KUKA KRL program: MyProgram_233().src

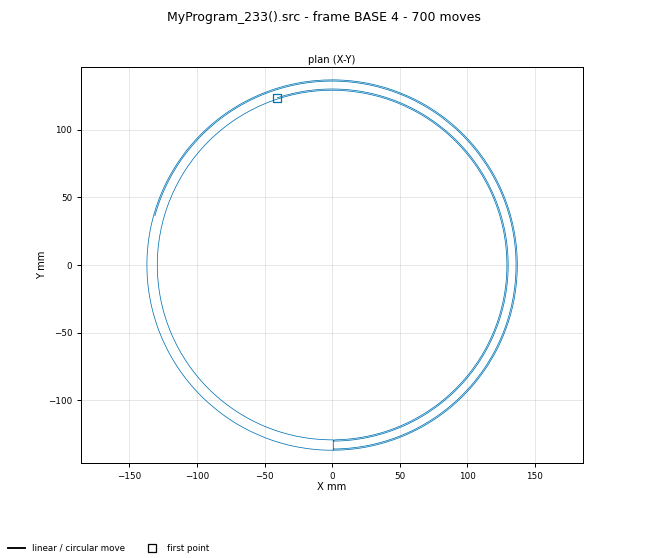
[picture p0: tool path of MyProgram_233().src in frame BASE 4, 700 of 700 moves have a stored position in this frame; points joined in program order, loops and branches not executed]
&ACCESS RVP
&REL 1
&PARAM TEMPLATE = C:\KRC\Roboter\Template\vorgabe
&PARAM EDITMASK = *
DEF MyProgram_233()
; ---- Setting reference (Base) ----
$BASE = BASE_DATA[4]

; --------------------------
; ---- Setting tool (TCP) ----
$TOOL = TOOL_DATA[3]
; --------------------------

$VEL.CP = VEL_APROX_PRINT
Startdeposition()
$VEL.CP = VEL_PRINT
LIN {X -40.5108,Y 123.8433,Z 158,A 106.7775,B 14.7751,C -0.259,E1 14.7289,E2 342.7672} C_DIS
LIN {X -37.5996,Y 124.7574,Z 158,A 105.4506,B 14.7751,C -0.2607,E1 14.7325,E2 344.0912} C_DIS
LIN {X -34.4379,Y 125.6675,Z 158,A 103.7953,B 14.7751,C -0.2561,E1 14.737,E2 345.7693} C_DIS
LIN {X -29.1894,Y 126.9876,Z 158,A 101.8109,B 14.7749,C -0.2693,E1 14.7422,E2 347.7066} C_DIS
LIN {X -26.9953,Y 127.473,Z 158,A 99.6139,B 14.7755,C -0.2357,E1 14.7486,E2 350.0402} C_DIS
LIN {X -20.6157,Y 128.6597,Z 158,A 97.7593,B 14.775,C -0.2658,E1 14.7534,E2 351.7799} C_DIS
LIN {X -13.8729,Y 129.5586,Z 158,A 94.7545,B 14.775,C -0.2668,E1 14.7617,E2 354.7844} C_DIS
LIN {X -10.0346,Y 129.9135,Z 158,A 93.1039,B 14.775,C -0.2686,E1 14.7663,E2 356.429} C_DIS
LIN {X -7.5089,Y 130.0837,Z 158,A 91.77,B 14.775,C -0.2625,E1 14.7701,E2 357.7876} C_DIS
LIN {X -2.8494,Y 130.27,Z 158,A 89.7989,B 14.775,C -0.2652,E1 14.7755,E2 359.7485} C_DIS
LIN {X 0.2302,Y 130.3001,Z 158,A 88.4188,B 14.775,C -0.2646,E1 14.7794,E2 361.131} C_DIS
LIN {X 4.1339,Y 130.2348,Z 158,A 86.7754,B 14.775,C -0.2668,E1 14.784,E2 362.7652} C_DIS
LIN {X 7.9856,Y 130.0543,Z 158,A 85.0604,B 14.775,C -0.2661,E1 14.7888,E2 364.4816} C_DIS
LIN {X 11.5872,Y 129.7845,Z 158,A 83.5435,B 14.775,C -0.268,E1 14.793,E2 365.9898} C_DIS
LIN {X 14.7399,Y 129.4647,Z 158,A 81.5298,B 14.7752,C -0.2493,E1 14.7987,E2 368.0739} C_DIS
LIN {X 19.1993,Y 128.8782,Z 158,A 80.1893,B 14.7749,C -0.2675,E1 14.8023,E2 369.341} C_DIS
LIN {X 22.8847,Y 128.2737,Z 158,A 78.3564,B 14.775,C -0.2612,E1 14.8073,E2 371.1953} C_DIS
LIN {X 27.0473,Y 127.4618,Z 158,A 76.5376,B 14.775,C -0.2616,E1 14.8123,E2 373.0085} C_DIS
LIN {X 30.989,Y 126.5612,Z 158,A 74.8488,B 14.775,C -0.2632,E1 14.8169,E2 374.6867} C_DIS
LIN {X 34.4256,Y 125.6709,Z 158,A 73.0922,B 14.7751,C -0.2562,E1 14.8217,E2 376.4656} C_DIS
LIN {X 37.7415,Y 124.7139,Z 158,A 71.8178,B 14.7751,C -0.2624,E1 14.825,E2 377.7118} C_DIS
LIN {X 41.1053,Y 123.6453,Z 158,A 70.2161,B 14.7751,C -0.2596,E1 14.8293,E2 379.3191} C_DIS
LIN {X 45.0082,Y 122.2809,Z 158,A 68.4489,B 14.7751,C -0.2595,E1 14.8339,E2 381.0806} C_DIS
LIN {X 47.9326,Y 121.1646,Z 158,A 67.0589,B 14.7751,C -0.2577,E1 14.8375,E2 382.4721} C_DIS
LIN {X 51.5684,Y 119.6599,Z 158,A 65.3226,B 14.7751,C -0.2556,E1 14.842,E2 384.2091} C_DIS
LIN {X 54.5031,Y 118.3521,Z 158,A 63.7925,B 14.7752,C -0.2504,E1 14.8459,E2 385.7528} C_DIS
LIN {X 58.0846,Y 116.637,Z 158,A 62.2133,B 14.7752,C -0.2534,E1 14.8498,E2 387.3129} C_DIS
LIN {X 60.819,Y 115.2341,Z 158,A 60.796,B 14.7752,C -0.2496,E1 14.8534,E2 388.738} C_DIS
LIN {X 63.7715,Y 113.6287,Z 158,A 59.2585,B 14.7753,C -0.2457,E1 14.8571,E2 390.2827} C_DIS
LIN {X 67.0742,Y 111.7117,Z 158,A 57.6957,B 14.7753,C -0.2469,E1 14.8609,E2 391.8325} C_DIS
LIN {X 70.2806,Y 109.722,Z 158,A 55.9342,B 14.7753,C -0.2412,E1 14.8651,E2 393.6062} C_DIS
LIN {X 74.0762,Y 107.1968,Z 158,A 54.0892,B 14.7753,C -0.2429,E1 14.8693,E2 395.4333} C_DIS
LIN {X 76.3123,Y 105.6161,Z 158,A 52.7396,B 14.7755,C -0.2364,E1 14.8724,E2 396.8001} C_DIS
LIN {X 83.8311,Y 99.7529,Z 158,A 48.7733,B 14.7755,C -0.2359,E1 14.8811,E2 400.7419} C_DIS
LIN {X 87.1361,Y 96.8796,Z 158,A 46.7285,B 14.7755,C -0.2285,E1 14.8854,E2 402.8014} C_DIS
LIN {X 90.1084,Y 94.121,Z 158,A 44.9408,B 14.7756,C -0.2248,E1 14.889,E2 404.5904} C_DIS
LIN {X 93.1997,Y 91.0613,Z 158,A 42.1103,B 14.7761,C -0.1919,E1 14.8947,E2 407.5274} C_DIS
LIN {X 97.7522,Y 86.1558,Z 158,A 40.368,B 14.7756,C -0.2235,E1 14.8977,E2 409.1333} C_DIS
LIN {X 99.829,Y 83.7404,Z 158,A 38.7374,B 14.7758,C -0.213,E1 14.9007,E2 410.7915} C_DIS
LIN {X 102.3423,Y 80.6497,Z 158,A 36.9316,B 14.7758,C -0.2073,E1 14.9039,E2 412.6046} C_DIS
LIN {X 105.1336,Y 76.9756,Z 158,A 35.0273,B 14.7758,C -0.2065,E1 14.9071,E2 414.4959} C_DIS
LIN {X 107.1572,Y 74.1333,Z 158,A 33.457,B 14.776,C -0.2017,E1 14.9096,E2 416.0716} C_DIS
LIN {X 109.47,Y 70.6733,Z 158,A 31.6182,B 14.776,C -0.1969,E1 14.9124,E2 417.9127} C_DIS
LIN {X 111.7477,Y 67.0138,Z 158,A 29.7051,B 14.776,C -0.1916,E1 14.9152,E2 419.8294} C_DIS
LIN {X 113.64,Y 63.7515,Z 158,A 28.0795,B 14.7761,C -0.1884,E1 14.9174,E2 421.4526} C_DIS
LIN {X 115.5412,Y 60.2341,Z 158,A 26.3549,B 14.7761,C -0.1849,E1 14.9197,E2 423.1746} C_DIS
LIN {X 117.1122,Y 57.1213,Z 158,A 24.9494,B 14.7761,C -0.1849,E1 14.9214,E2 424.5666} C_DIS
LIN {X 118.4334,Y 54.3273,Z 158,A 23.5787,B 14.7762,C -0.1809,E1 14.9231,E2 425.9399} C_DIS
LIN {X 119.9368,Y 50.927,Z 158,A 21.9716,B 14.7762,C -0.1774,E1 14.9248,E2 427.5454} C_DIS
LIN {X 121.0941,Y 48.1087,Z 158,A 20.662,B 14.7762,C -0.1747,E1 14.9262,E2 428.8527} C_DIS
LIN {X 122.0988,Y 45.4943,Z 158,A 19.4496,B 14.7763,C -0.1719,E1 14.9274,E2 430.0639} C_DIS
LIN {X 123.1367,Y 42.6048,Z 158,A 18.0772,B 14.7763,C -0.1674,E1 14.9287,E2 431.4403} C_DIS
LIN {X 124.1541,Y 39.5421,Z 158,A 16.6266,B 14.7764,C -0.1623,E1 14.9299,E2 432.896} C_DIS
LIN {X 125.2221,Y 36.0224,Z 158,A 15.079,B 14.7764,C -0.16,E1 14.9312,E2 434.4372} C_DIS
LIN {X 126.1859,Y 32.4831,Z 158,A 13.215,B 14.7766,C -0.1471,E1 14.9325,E2 436.3323} C_DIS
LIN {X 127.3684,Y 27.4799,Z 158,A 10.9043,B 14.7766,C -0.1389,E1 14.9339,E2 438.6511} C_DIS
LIN {X 128.028,Y 24.2226,Z 158,A 9.7326,B 14.7766,C -0.1441,E1 14.9345,E2 439.7907} C_DIS
LIN {X 128.6085,Y 20.928,Z 158,A 7.975,B 14.7767,C -0.1304,E1 14.9354,E2 441.5834} C_DIS
LIN {X 129.1193,Y 17.5046,Z 158,A 6.6957,B 14.7767,C -0.1338,E1 14.9358,E2 442.8361} C_DIS
LIN {X 129.5993,Y 13.4944,Z 158,A 5.074,B 14.7767,C -0.1336,E1 14.9363,E2 444.4418} C_DIS
LIN {X 129.9364,Y 9.7203,Z 158,A 3.3807,B 14.7767,C -0.1277,E1 14.9367,E2 446.1402} C_DIS
LIN {X 130.1635,Y 5.9747,Z 158,A 1.6403,B 14.7768,C -0.1198,E1 14.937,E2 447.8932} C_DIS
LIN {X 130.2801,Y 2.244,Z 158,A 0.1423,B 14.7768,C -0.1196,E1 14.937,E2 449.3764} C_DIS
LIN {X 130.2859,Y -1.8955,Z 158,A -1.6435,B 14.7768,C -0.1152,E1 14.937,E2 451.1603} C_DIS
LIN {X 130.19,Y -5.3434,Z 158,A -3.2527,B 14.7769,C -0.1076,E1 14.937,E2 452.7822} C_DIS
LIN {X 129.9186,Y -9.9649,Z 158,A -5.9348,B 14.7771,C -0.0802,E1 14.9364,E2 455.5425} C_DIS
LIN {X 129.3731,Y -15.5074,Z 158,A -7.5578,B 14.777,C -0.1,E1 14.9359,E2 457.0719} C_DIS
LIN {X 129.005,Y -18.3195,Z 158,A -9.5341,B 14.7771,C -0.0723,E1 14.9351,E2 459.1353} C_DIS
LIN {X 128.1366,Y -23.6512,Z 158,A -11.1383,B 14.7771,C -0.0905,E1 14.9343,E2 460.6523} C_DIS
LIN {X 127.2398,Y -28.0756,Z 158,A -13.1387,B 14.7771,C -0.0841,E1 14.9332,E2 462.6571} C_DIS
LIN {X 126.2536,Y -32.2163,Z 158,A -15.0385,B 14.7771,C -0.0776,E1 14.9319,E2 464.5625} C_DIS
LIN {X 124.8734,Y -37.2135,Z 158,A -17.2259,B 14.7771,C -0.0739,E1 14.9302,E2 466.7422} C_DIS
LIN {X 123.7298,Y -40.8516,Z 158,A -18.9168,B 14.7771,C -0.0686,E1 14.9288,E2 468.4368} C_DIS
LIN {X 122.6296,Y -44.0434,Z 158,A -21.7356,B 14.7773,C -0.0208,E1 14.926,E2 471.4133} C_DIS
LIN {X 119.44,Y -52.0772,Z 158,A -24.233,B 14.7773,C -0.0524,E1 14.9234,E2 473.7638} C_DIS
LIN {X 116.7284,Y -57.8993,Z 158,A -27.0512,B 14.7773,C -0.0448,E1 14.92,E2 476.585} C_DIS
LIN {X 114.986,Y -61.2914,Z 158,A -28.6247,B 14.7773,C -0.0436,E1 14.918,E2 478.1486} C_DIS
LIN {X 112.9775,Y -64.9195,Z 158,A -30.4029,B 14.7773,C -0.0402,E1 14.9156,E2 479.9238} C_DIS
LIN {X 110.9729,Y -68.2886,Z 158,A -32.0131,B 14.7773,C -0.0393,E1 14.9133,E2 481.5227} C_DIS
LIN {X 109.6462,Y -70.3989,Z 158,A -33.112,B 14.7773,C -0.0363,E1 14.9116,E2 482.6234} C_DIS
LIN {X 108.2654,Y -72.5046,Z 158,A -34.3195,B 14.7773,C -0.0302,E1 14.9097,E2 483.8442} C_DIS
LIN {X 105.9657,Y -75.8258,Z 158,A -36.2678,B 14.7773,C -0.0201,E1 14.9066,E2 485.8151} C_DIS
LIN {X 103.7855,Y -78.7844,Z 158,A -37.7168,B 14.7773,C -0.0215,E1 14.9042,E2 487.2465} C_DIS
LIN {X 101.3531,Y -81.8892,Z 158,A -39.4296,B 14.7773,C -0.0179,E1 14.9012,E2 488.9589} C_DIS
LIN {X 98.3316,Y -85.494,Z 158,A -41.7666,B 14.7773,C -0.0043,E1 14.8969,E2 491.3301} C_DIS
LIN {X 96.0761,Y -88.0211,Z 158,A -42.911,B 14.7773,C -0.012,E1 14.8948,E2 492.4356} C_DIS
LIN {X 93.3589,Y -90.8985,Z 158,A -44.7247,B 14.7773,C -0.0056,E1 14.8913,E2 494.2602} C_DIS
LIN {X 89.4912,Y -94.7081,Z 158,A -47.1654,B 14.7773,C 0.0013,E1 14.8864,E2 496.71} C_DIS
LIN {X 86.752,Y -97.2236,Z 158,A -48.7508,B 14.7773,C 0.0032,E1 14.8831,E2 498.2915} C_DIS
LIN {X 83.627,Y -99.9241,Z 158,A -50.4995,B 14.7773,C 0.0048,E1 14.8794,E2 500.0343} C_DIS
LIN {X 80.0007,Y -102.8504,Z 158,A -52.3931,B 14.7773,C 0.0039,E1 14.8753,E2 501.9119} C_DIS
LIN {X 78.0349,Y -104.3499,Z 158,A -53.5757,B 14.7773,C 0.0091,E1 14.8726,E2 503.107} C_DIS
LIN {X 75.6115,Y -106.119,Z 158,A -54.8753,B 14.7773,C 0.0109,E1 14.8697,E2 504.4058} C_DIS
LIN {X 72.5816,Y -108.214,Z 158,A -56.3904,B 14.7773,C 0.0105,E1 14.8662,E2 505.9102} C_DIS
LIN {X 70.5262,Y -109.5648,Z 158,A -57.4656,B 14.7773,C 0.0122,E1 14.8637,E2 506.9858} C_DIS
LIN {X 67.235,Y -111.6145,Z 158,A -59.2828,B 14.7773,C 0.0187,E1 14.8593,E2 508.8182} C_DIS
LIN {X 63.65,Y -113.697,Z 158,A -61.5059,B 14.7773,C 0.0343,E1 14.8538,E2 511.0903} C_DIS
LIN {X 60.2129,Y -115.5523,Z 158,A -63.3497,B 14.7773,C 0.0409,E1 14.8492,E2 512.9505} C_DIS
LIN {X 56.033,Y -117.6355,Z 158,A -64.8162,B 14.7773,C 0.0254,E1 14.8457,E2 514.3499} C_DIS
LIN {X 52.9667,Y -119.0478,Z 158,A -66.328,B 14.7773,C 0.0283,E1 14.8418,E2 515.8664} C_DIS
LIN {X 49.793,Y -120.4103,Z 158,A -67.7428,B 14.7773,C 0.027,E1 14.8382,E2 517.2703} C_DIS
LIN {X 46.482,Y -121.7285,Z 158,A -69.3474,B 14.7773,C 0.0302,E1 14.834,E2 518.8807} C_DIS
LIN {X 43.6924,Y -122.7561,Z 158,A -70.6467,B 14.7773,C 0.0314,E1 14.8306,E2 520.1802} C_DIS
LIN {X 37.793,Y -124.6982,Z 158,A -73.2996,B 14.7773,C 0.0319,E1 14.8236,E2 522.8262} C_DIS
LIN {X 34.1254,Y -125.7522,Z 158,A -74.9414,B 14.7773,C 0.0324,E1 14.8192,E2 524.465} C_DIS
LIN {X 31.4215,Y -126.4553,Z 158,A -76.5158,B 14.7773,C 0.0442,E1 14.8148,E2 526.0813} C_DIS
LIN {X 24.1591,Y -128.0402,Z 158,A -79.544,B 14.7773,C 0.0393,E1 14.8066,E2 529.0834} C_DIS
LIN {X 21.0197,Y -128.5932,Z 158,A -80.9175,B 14.7773,C 0.0393,E1 14.8028,E2 530.4546} C_DIS
LIN {X 17.736,Y -129.0883,Z 158,A -82.5197,B 14.7773,C 0.0446,E1 14.7983,E2 532.0746} C_DIS
LIN {X 13.8148,Y -129.5649,Z 158,A -84.1828,B 14.7773,C 0.0432,E1 14.7937,E2 533.73} C_DIS
LIN {X 9.1695,Y -129.9766,Z 158,A -86.2845,B 14.7773,C 0.0455,E1 14.7879,E2 535.8389} C_DIS
LIN {X 5.0148,Y -130.2028,Z 158,A -88.0308,B 14.7773,C 0.0436,E1 14.783,E2 537.5764} C_DIS
LIN {X 0.9154,Y -130.2963,Z 158,A -89.8605,B 14.7773,C 0.0447,E1 14.7779,E2 539.4102} C_DIS
Enddeposition()
LIN {X 0.9154,Y -130.2963,Z 158,A -89.8605,B 14.7773,C 0.0447,E1 14.7779,E2 539.4102} C_DIS
Startdeposition()
$VEL.CP = VEL_PRINT
LIN {X 1.8704,Y -129.3568,Z 158,A -88.8345,B 14.7779,C 0.0171,E1 14.7817,E2 538.2762} C_DIS
LIN {X 5.0391,Y -129.2718,Z 158,A -87.4155,B 14.7779,C 0.0163,E1 14.7857,E2 536.8546} C_DIS
LIN {X 7.9326,Y -129.1265,Z 158,A -86.0775,B 14.7779,C 0.0142,E1 14.7894,E2 535.5095} C_DIS
LIN {X 11.1084,Y -128.8923,Z 158,A -84.6755,B 14.7779,C 0.0139,E1 14.7933,E2 534.1076} C_DIS
LIN {X 14.2559,Y -128.5827,Z 158,A -83.1246,B 14.7779,C 0.0087,E1 14.7977,E2 532.538} C_DIS
LIN {X 17.4162,Y -128.1936,Z 158,A -81.876,B 14.7779,C 0.0129,E1 14.8011,E2 531.3078} C_DIS
LIN {X 20.566,Y -127.7268,Z 158,A -80.3675,B 14.7779,C 0.009,E1 14.8053,E2 529.7867} C_DIS
LIN {X 24.2361,Y -127.0793,Z 158,A -78.992,B 14.7779,C 0.0163,E1 14.809,E2 528.4426} C_DIS
LIN {X 26.7211,Y -126.5815,Z 158,A -77.7134,B 14.7779,C 0.0107,E1 14.8125,E2 527.1448} C_DIS
LIN {X 29.9082,Y -125.8658,Z 158,A -76.181,B 14.7779,C 0.0068,E1 14.8167,E2 525.601} C_DIS
LIN {X 33.2672,Y -125.0192,Z 158,A -74.8008,B 14.7779,C 0.0102,E1 14.8204,E2 524.2379} C_DIS
LIN {X 36.0209,Y -124.2542,Z 158,A -73.4572,B 14.7779,C 0.0065,E1 14.824,E2 522.884} C_DIS
LIN {X 39.0482,Y -123.3363,Z 158,A -72.0632,B 14.7779,C 0.0053,E1 14.8278,E2 521.4897} C_DIS
LIN {X 42.4611,Y -122.2029,Z 158,A -70.5633,B 14.7779,C 0.0064,E1 14.8317,E2 519.9994} C_DIS
LIN {X 45.0721,Y -121.2646,Z 158,A -69.2472,B 14.7779,C 0.0023,E1 14.8352,E2 518.672} C_DIS
LIN {X 48.0423,Y -120.1189,Z 158,A -67.8483,B 14.7779,C 0.0008,E1 14.8388,E2 517.273} C_DIS
LIN {X 50.972,Y -118.9054,Z 158,A -66.4449,B 14.7779,C -0.001,E1 14.8424,E2 515.8685} C_DIS
LIN {X 53.8674,Y -117.6222,Z 158,A -65.063,B 14.7779,C -0.0022,E1 14.8459,E2 514.4877} C_DIS
LIN {X 56.6975,Y -116.285,Z 158,A -63.6928,B 14.7779,C -0.0037,E1 14.8494,E2 513.1181} C_DIS
LIN {X 59.4453,Y -114.9057,Z 158,A -62.3199,B 14.7779,C -0.0061,E1 14.8528,E2 511.7426} C_DIS
LIN {X 62.4679,Y -113.2907,Z 158,A -60.7953,B 14.7779,C -0.0087,E1 14.8566,E2 510.2156} C_DIS
LIN {X 65.1434,Y -111.7741,Z 158,A -59.4503,B 14.7779,C -0.0104,E1 14.8598,E2 508.8712} C_DIS
LIN {X 68.4953,Y -109.7515,Z 158,A -57.8772,B 14.7779,C -0.0082,E1 14.8635,E2 507.3155} C_DIS
LIN {X 70.5632,Y -108.4335,Z 158,A -56.6501,B 14.7779,C -0.0146,E1 14.8664,E2 506.0704} C_DIS
LIN {X 73.1984,Y -106.6722,Z 158,A -55.2581,B 14.7779,C -0.0168,E1 14.8697,E2 504.6782} C_DIS
LIN {X 75.7896,Y -104.8472,Z 158,A -53.8699,B 14.7779,C -0.0189,E1 14.8728,E2 503.2903} C_DIS
LIN {X 78.9589,Y -102.4822,Z 158,A -51.9922,B 14.7779,C -0.0264,E1 14.877,E2 501.3956} C_DIS
LIN {X 82.0782,Y -100.001,Z 158,A -50.2104,B 14.7779,C -0.0305,E1 14.8809,E2 499.6098} C_DIS
LIN {X 85.6925,Y -96.9214,Z 158,A -48.1287,B 14.7779,C -0.0342,E1 14.8853,E2 497.5282} C_DIS
LIN {X 89.1886,Y -93.7146,Z 158,A -46.1035,B 14.7779,C -0.0363,E1 14.8894,E2 495.5096} C_DIS
LIN {X 92.0419,Y -90.9142,Z 158,A -44.279,B 14.7779,C -0.042,E1 14.893,E2 493.6765} C_DIS
LIN {X 95.313,Y -87.478,Z 158,A -42.2006,B 14.7779,C -0.0461,E1 14.897,E2 491.5983} C_DIS
LIN {X 98.4499,Y -83.9322,Z 158,A -40.2684,B 14.7779,C -0.0457,E1 14.9005,E2 489.6831} C_DIS
LIN {X 101.0061,Y -80.8384,Z 158,A -38.36,B 14.7779,C -0.0543,E1 14.9039,E2 487.7568} C_DIS
LIN {X 103.901,Y -77.0817,Z 158,A -36.4277,B 14.7779,C -0.054,E1 14.9071,E2 485.8419} C_DIS
LIN {X 105.7745,Y -74.4898,Z 158,A -35.026,B 14.7779,C -0.0571,E1 14.9094,E2 484.4401} C_DIS
LIN {X 107.5679,Y -71.8758,Z 158,A -33.6347,B 14.7778,C -0.0603,E1 14.9116,E2 483.0485} C_DIS
LIN {X 109.2967,Y -69.2188,Z 158,A -32.2315,B 14.7778,C -0.0639,E1 14.9137,E2 481.6435} C_DIS
LIN {X 110.9657,Y -66.5108,Z 158,A -30.8514,B 14.7778,C -0.0667,E1 14.9157,E2 480.265} C_DIS
LIN {X 112.5675,Y -63.7628,Z 158,A -29.4479,B 14.7778,C -0.0703,E1 14.9176,E2 478.8604} C_DIS
LIN {X 114.1018,Y -60.974,Z 158,A -28.0337,B 14.7778,C -0.0743,E1 14.9195,E2 477.4438} C_DIS
LIN {X 115.5605,Y -58.1599,Z 158,A -26.5379,B 14.7778,C -0.0812,E1 14.9214,E2 475.9351} C_DIS
LIN {X 116.9596,Y -55.2918,Z 158,A -25.208,B 14.7777,C -0.0824,E1 14.923,E2 474.6133} C_DIS
LIN {X 118.2696,Y -52.4305,Z 158,A -23.8839,B 14.7777,C -0.084,E1 14.9245,E2 473.2957} C_DIS
LIN {X 119.5144,Y -49.5268,Z 158,A -22.4999,B 14.7777,C -0.0874,E1 14.926,E2 471.9116} C_DIS
LIN {X 120.6905,Y -46.5873,Z 158,A -21.1146,B 14.7777,C -0.0909,E1 14.9275,E2 470.5265} C_DIS
LIN {X 121.8119,Y -43.5713,Z 158,A -19.7027,B 14.7777,C -0.0946,E1 14.9288,E2 469.1143} C_DIS
LIN {X 122.8405,Y -40.5809,Z 158,A -18.3158,B 14.7777,C -0.0982,E1 14.93,E2 467.7271} C_DIS
LIN {X 123.798,Y -37.5587,Z 158,A -16.9229,B 14.7776,C -0.1019,E1 14.9312,E2 466.3337} C_DIS
LIN {X 124.6862,Y -34.4963,Z 158,A -15.4594,B 14.7776,C -0.1077,E1 14.9323,E2 464.8624} C_DIS
LIN {X 125.6787,Y -30.6845,Z 158,A -13.9628,B 14.7776,C -0.1047,E1 14.9333,E2 463.3928} C_DIS
LIN {X 126.2253,Y -28.3536,Z 158,A -12.7571,B 14.7775,C -0.1126,E1 14.9341,E2 462.1686} C_DIS
LIN {X 126.9119,Y -25.1076,Z 158,A -11.3092,B 14.7775,C -0.1163,E1 14.9349,E2 460.7213} C_DIS
LIN {X 127.464,Y -22.1343,Z 158,A -9.9823,B 14.7775,C -0.1199,E1 14.9355,E2 459.3942} C_DIS
LIN {X 127.9772,Y -18.9423,Z 158,A -8.5548,B 14.7775,C -0.124,E1 14.9362,E2 457.9653} C_DIS
LIN {X 128.394,Y -15.8699,Z 158,A -7.2017,B 14.7774,C -0.1275,E1 14.9366,E2 456.6129} C_DIS
LIN {X 128.732,Y -12.8404,Z 158,A -5.8713,B 14.7774,C -0.1309,E1 14.937,E2 455.283} C_DIS
LIN {X 129.0205,Y -9.5023,Z 158,A -4.391,B 14.7774,C -0.1353,E1 14.9374,E2 453.8013} C_DIS
LIN {X 129.2548,Y -5.4753,Z 158,A -2.5487,B 14.7772,C -0.1425,E1 14.9376,E2 451.9502} C_DIS
LIN {X 129.3623,Y -1.5416,Z 158,A -0.9468,B 14.7772,C -0.1431,E1 14.9377,E2 450.3629} C_DIS
LIN {X 129.3615,Y 1.5923,Z 158,A 0.493,B 14.7772,C -0.149,E1 14.9377,E2 448.9152} C_DIS
LIN {X 129.2822,Y 4.773,Z 158,A 2.0333,B 14.7771,C -0.1576,E1 14.9375,E2 447.3576} C_DIS
LIN {X 129.0371,Y 9.2755,Z 158,A 3.8932,B 14.7771,C -0.159,E1 14.9372,E2 445.5116} C_DIS
LIN {X 128.7458,Y 12.6969,Z 158,A 5.4984,B 14.7771,C -0.1664,E1 14.9368,E2 443.8947} C_DIS
LIN {X 128.3979,Y 15.837,Z 158,A 6.7268,B 14.7771,C -0.1649,E1 14.9364,E2 442.6848} C_DIS
LIN {X 127.9661,Y 19.02,Z 158,A 8.1441,B 14.777,C -0.1689,E1 14.9358,E2 441.2666} C_DIS
LIN {X 127.4679,Y 22.1126,Z 158,A 9.5203,B 14.777,C -0.1726,E1 14.9352,E2 439.8902} C_DIS
LIN {X 126.8921,Y 25.2051,Z 158,A 10.8943,B 14.7769,C -0.1761,E1 14.9345,E2 438.5168} C_DIS
LIN {X 126.2078,Y 28.4299,Z 158,A 12.272,B 14.7769,C -0.1777,E1 14.9337,E2 437.1471} C_DIS
LIN {X 125.489,Y 31.451,Z 158,A 13.7046,B 14.7769,C -0.1835,E1 14.9327,E2 435.7064} C_DIS
LIN {X 124.6841,Y 34.5036,Z 158,A 15.2093,B 14.7767,C -0.1911,E1 14.9316,E2 434.1876} C_DIS
LIN {X 123.7981,Y 37.5584,Z 158,A 16.4848,B 14.7767,C -0.1907,E1 14.9306,E2 432.9264} C_DIS
LIN {X 122.8363,Y 40.5934,Z 158,A 17.9865,B 14.7767,C -0.1977,E1 14.9293,E2 431.4124} C_DIS
LIN {X 121.8029,Y 43.5963,Z 158,A 19.2664,B 14.7767,C -0.1975,E1 14.9281,E2 430.1461} C_DIS
LIN {X 120.6965,Y 46.5719,Z 158,A 20.6608,B 14.7766,C -0.201,E1 14.9267,E2 428.7516} C_DIS
LIN {X 119.518,Y 49.5181,Z 158,A 22.052,B 14.7766,C -0.2044,E1 14.9253,E2 427.3608} C_DIS
LIN {X 118.2648,Y 52.4412,Z 158,A 23.4461,B 14.7765,C -0.2078,E1 14.9237,E2 425.9671} C_DIS
LIN {X 116.9451,Y 55.3221,Z 158,A 24.8349,B 14.7765,C -0.2111,E1 14.9221,E2 424.5787} C_DIS
LIN {X 115.5543,Y 58.1721,Z 158,A 26.2245,B 14.7765,C -0.2143,E1 14.9203,E2 423.1897} C_DIS
LIN {X 113.9971,Y 61.1689,Z 158,A 27.6625,B 14.7764,C -0.2163,E1 14.9185,E2 421.7571} C_DIS
LIN {X 112.5602,Y 63.7755,Z 158,A 29.0181,B 14.7764,C -0.2209,E1 14.9166,E2 420.3962} C_DIS
LIN {X 110.9695,Y 66.5044,Z 158,A 30.4133,B 14.7763,C -0.2244,E1 14.9146,E2 419.0002} C_DIS
LIN {X 108.9939,Y 69.6944,Z 158,A 31.9443,B 14.7763,C -0.2243,E1 14.9124,E2 417.4832} C_DIS
LIN {X 107.5569,Y 71.8922,Z 158,A 33.2084,B 14.7762,C -0.2304,E1 14.9104,E2 416.2064} C_DIS
LIN {X 105.7623,Y 74.507,Z 158,A 34.5986,B 14.7762,C -0.2333,E1 14.9082,E2 414.8169} C_DIS
LIN {X 103.5733,Y 77.5218,Z 158,A 36.2797,B 14.776,C -0.2382,E1 14.9054,E2 413.131} C_DIS
LIN {X 101.0079,Y 80.8362,Z 158,A 38.24,B 14.776,C -0.2458,E1 14.902,E2 411.1573} C_DIS
LIN {X 97.9574,Y 84.5063,Z 158,A 40.175,B 14.776,C -0.2448,E1 14.8985,E2 409.2418} C_DIS
LIN {X 95.8745,Y 86.8623,Z 158,A 41.7048,B 14.7758,C -0.2522,E1 14.8957,E2 407.6953} C_DIS
LIN {X 92.6666,Y 90.2775,Z 158,A 43.7557,B 14.7758,C -0.2558,E1 14.8917,E2 405.646} C_DIS
LIN {X 89.7778,Y 93.1504,Z 158,A 45.5701,B 14.7757,C -0.2598,E1 14.8881,E2 403.8295} C_DIS
LIN {X 86.2924,Y 96.3877,Z 158,A 47.6586,B 14.7757,C -0.2633,E1 14.8838,E2 401.7421} C_DIS
LIN {X 83.298,Y 98.9871,Z 158,A 49.3903,B 14.7756,C -0.2659,E1 14.8801,E2 400.0126} C_DIS
LIN {X 79.6543,Y 101.9424,Z 158,A 51.3138,B 14.7756,C -0.2647,E1 14.8759,E2 398.1063} C_DIS
LIN {X 76.5448,Y 104.297,Z 158,A 52.8952,B 14.7756,C -0.2631,E1 14.8724,E2 396.5412} C_DIS
LIN {X 74.494,Y 105.7716,Z 158,A 54.141,B 14.7756,C -0.269,E1 14.8696,E2 395.2803} C_DIS
LIN {X 71.8789,Y 107.5658,Z 158,A 55.5369,B 14.7755,C -0.271,E1 14.8663,E2 393.885} C_DIS
LIN {X 68.5385,Y 109.7246,Z 158,A 57.4465,B 14.7754,C -0.2783,E1 14.8618,E2 391.9577} C_DIS
LIN {X 65.138,Y 111.7772,Z 158,A 59.0374,B 14.7754,C -0.2756,E1 14.858,E2 390.386} C_DIS
LIN {X 62.3796,Y 113.3396,Z 158,A 60.4418,B 14.7754,C -0.2775,E1 14.8546,E2 388.9813} C_DIS
LIN {X 59.5725,Y 114.839,Z 158,A 61.8465,B 14.7754,C -0.2793,E1 14.8511,E2 387.577} C_DIS
LIN {X 56.7398,Y 116.2642,Z 158,A 63.2428,B 14.7754,C -0.2808,E1 14.8476,E2 386.1814} C_DIS
LIN {X 53.873,Y 117.6196,Z 158,A 64.6388,B 14.7753,C -0.2822,E1 14.8441,E2 384.7862} C_DIS
LIN {X 50.6665,Y 119.0375,Z 158,A 66.1801,B 14.7753,C -0.2835,E1 14.8401,E2 383.2463} C_DIS
LIN {X 48.0346,Y 120.1219,Z 158,A 67.4419,B 14.7753,C -0.2849,E1 14.8369,E2 381.9843} C_DIS
LIN {X 45.0726,Y 121.2644,Z 158,A 68.8419,B 14.7753,C -0.2861,E1 14.8332,E2 380.5849} C_DIS
LIN {X 41.276,Y 122.609,Z 158,A 70.79,B 14.7751,C -0.2927,E1 14.828,E2 378.6179} C_DIS
LIN {X 37.5536,Y 123.7995,Z 158,A 72.3454,B 14.7751,C -0.2888,E1 14.8239,E2 377.083} C_DIS
LIN {X 34.5005,Y 124.685,Z 158,A 73.824,B 14.7751,C -0.2919,E1 14.8199,E2 375.5964} C_DIS
LIN {X 30.8477,Y 125.6393,Z 158,A 75.3196,B 14.7751,C -0.2877,E1 14.816,E2 374.1214} C_DIS
LIN {X 28.3547,Y 126.225,Z 158,A 76.543,B 14.7751,C -0.291,E1 14.8126,E2 372.888} C_DIS
LIN {X 25.2462,Y 126.8837,Z 158,A 77.9451,B 14.7751,C -0.2916,E1 14.8088,E2 371.4868} C_DIS
LIN {X 22.1444,Y 127.4622,Z 158,A 79.4205,B 14.7751,C -0.2945,E1 14.8047,E2 370.0029} C_DIS
LIN {X 18.985,Y 127.9711,Z 158,A 80.8587,B 14.7751,C -0.2957,E1 14.8007,E2 368.5626} C_DIS
LIN {X 15.883,Y 128.3924,Z 158,A 82.1755,B 14.7751,C -0.294,E1 14.7971,E2 367.2542} C_DIS
LIN {X 12.6795,Y 128.7475,Z 158,A 83.5848,B 14.7751,C -0.2938,E1 14.7932,E2 365.8475} C_DIS
LIN {X 9.5064,Y 129.0202,Z 158,A 85.1433,B 14.775,C -0.2984,E1 14.7888,E2 364.2725} C_DIS
LIN {X 5.4109,Y 129.2573,Z 158,A 86.9292,B 14.775,C -0.2976,E1 14.7838,E2 362.491} C_DIS
LIN {X 1.5855,Y 129.3616,Z 158,A 88.4775,B 14.775,C -0.2932,E1 14.7795,E2 360.9603} C_DIS
LIN {X -1.5842,Y 129.3616,Z 158,A 89.9211,B 14.775,C -0.2942,E1 14.7755,E2 359.5128} C_DIS
LIN {X -4.768,Y 129.2824,Z 158,A 91.4165,B 14.775,C -0.2964,E1 14.7713,E2 358.0083} C_DIS
LIN {X -7.9373,Y 129.1262,Z 158,A 92.719,B 14.775,C -0.2931,E1 14.7677,E2 356.7183} C_DIS
LIN {X -11.1107,Y 128.8921,Z 158,A 94.1241,B 14.775,C -0.2925,E1 14.7638,E2 355.3146} C_DIS
LIN {X -15.0056,Y 128.4971,Z 158,A 95.6793,B 14.7752,C -0.2866,E1 14.7595,E2 353.7809} C_DIS
LIN {X -17.4315,Y 128.1916,Z 158,A 96.9383,B 14.7752,C -0.2911,E1 14.756,E2 352.5025} C_DIS
LIN {X -20.558,Y 127.7281,Z 158,A 98.3577,B 14.7752,C -0.2909,E1 14.7521,E2 351.0817} C_DIS
LIN {X -23.648,Y 127.1917,Z 158,A 99.7546,B 14.7752,C -0.2903,E1 14.7482,E2 349.6849} C_DIS
LIN {X -26.8057,Y 126.5632,Z 158,A 101.1804,B 14.7752,C -0.2893,E1 14.7443,E2 348.2601} C_DIS
LIN {X -29.8929,Y 125.8695,Z 158,A 102.5896,B 14.7752,C -0.2885,E1 14.7405,E2 346.8509} C_DIS
LIN {X -32.9844,Y 125.0947,Z 158,A 104.1378,B 14.7752,C -0.2912,E1 14.7363,E2 345.2881} C_DIS
LIN {X -36.0387,Y 124.249,Z 158,A 105.4058,B 14.7752,C -0.286,E1 14.7329,E2 344.0368} C_DIS
LIN {X -39.0711,Y 123.329,Z 158,A 106.8132,B 14.7752,C -0.2848,E1 14.7292,E2 342.63} C_DIS
LIN {X -42.071,Y 122.3381,Z 158,A 108.2261,B 14.7752,C -0.2837,E1 14.7254,E2 341.2168} C_DIS
LIN {X -45.0765,Y 121.2629,Z 158,A 109.6389,B 14.7752,C -0.2821,E1 14.7217,E2 339.8053} C_DIS
LIN {X -48.0477,Y 120.1167,Z 158,A 111.0564,B 14.7753,C -0.2806,E1 14.7181,E2 338.3882} C_DIS
LIN {X -50.9916,Y 118.8969,Z 158,A 112.4639,B 14.7753,C -0.2787,E1 14.7144,E2 336.9825} C_DIS
LIN {X -53.877,Y 117.6178,Z 158,A 114.001,B 14.7753,C -0.2808,E1 14.7105,E2 335.4307} C_DIS
LIN {X -56.7409,Y 116.2636,Z 158,A 115.2781,B 14.7754,C -0.2753,E1 14.7073,E2 334.1694} C_DIS
LIN {X -59.5696,Y 114.8405,Z 158,A 116.6737,B 14.7754,C -0.2731,E1 14.7038,E2 332.7759} C_DIS
LIN {X -62.9274,Y 113.0363,Z 158,A 118.2492,B 14.7756,C -0.2674,E1 14.7,E2 331.2151} C_DIS
LIN {X -65.1416,Y 111.7752,Z 158,A 119.5345,B 14.7756,C -0.2699,E1 14.6969,E2 329.913} C_DIS
LIN {X -67.8877,Y 110.1286,Z 158,A 120.9556,B 14.7756,C -0.2677,E1 14.6935,E2 328.493} C_DIS
LIN {X -70.5661,Y 108.4316,Z 158,A 122.368,B 14.7756,C -0.2655,E1 14.6902,E2 327.0811} C_DIS
LIN {X -73.2027,Y 106.6693,Z 158,A 123.778,B 14.7756,C -0.2632,E1 14.6869,E2 325.672} C_DIS
LIN {X -76.1949,Y 104.5534,Z 158,A 125.3216,B 14.7757,C -0.258,E1 14.6834,E2 324.1393} C_DIS
LIN {X -78.9664,Y 102.4763,Z 158,A 126.956,B 14.7757,C -0.2579,E1 14.6798,E2 322.4951} C_DIS
LIN {X -82.0795,Y 100,Z 158,A 128.8942,B 14.7757,C -0.2592,E1 14.6755,E2 320.5386} C_DIS
LIN {X -85.6992,Y 96.9154,Z 158,A 131.0102,B 14.7757,C -0.2552,E1 14.6711,E2 318.424} C_DIS
LIN {X -89.2031,Y 93.7008,Z 158,A 132.9715,B 14.7759,C -0.2468,E1 14.6671,E2 316.4817} C_DIS
LIN {X -91.4858,Y 91.4739,Z 158,A 134.5617,B 14.7759,C -0.2485,E1 14.6639,E2 314.8728} C_DIS
LIN {X -94.7812,Y 88.054,Z 158,A 136.6786,B 14.7759,C -0.2441,E1 14.6598,E2 312.7569} C_DIS
LIN {X -97.9529,Y 84.5116,Z 158,A 138.6439,B 14.7761,C -0.2355,E1 14.6563,E2 310.8103} C_DIS
LIN {X -100.5113,Y 81.4526,Z 158,A 140.5743,B 14.7761,C -0.2357,E1 14.6528,E2 308.8633} C_DIS
LIN {X -102.9643,Y 78.329,Z 158,A 142.2007,B 14.7762,C -0.2278,E1 14.6501,E2 307.2543} C_DIS
LIN {X -104.8445,Y 75.7932,Z 158,A 143.7391,B 14.7762,C -0.2281,E1 14.6475,E2 305.7015} C_DIS
LIN {X -106.6807,Y 73.186,Z 158,A 145.032,B 14.7762,C -0.2213,E1 14.6455,E2 304.4241} C_DIS
LIN {X -108.4481,Y 70.5408,Z 158,A 146.4491,B 14.7763,C -0.2179,E1 14.6433,E2 303.0078} C_DIS
LIN {X -110.1463,Y 67.8588,Z 158,A 147.8684,B 14.7763,C -0.2146,E1 14.6412,E2 301.5888} C_DIS
LIN {X -112.1734,Y 64.4535,Z 158,A 149.7961,B 14.7763,C -0.2146,E1 14.6384,E2 299.6436} C_DIS
LIN {X -114.2931,Y 60.612,Z 158,A 151.6317,B 14.7765,C -0.2065,E1 14.636,E2 297.8228} C_DIS
LIN {X -115.5666,Y 58.1479,Z 158,A 152.8531,B 14.7765,C -0.2029,E1 14.6345,E2 296.6038} C_DIS
LIN {X -116.9562,Y 55.299,Z 158,A 154.2861,B 14.7765,C -0.1998,E1 14.6328,E2 295.1693} C_DIS
LIN {X -118.2711,Y 52.427,Z 158,A 155.68,B 14.7767,C -0.1958,E1 14.6312,E2 293.7778} C_DIS
LIN {X -119.5204,Y 49.5126,Z 158,A 157.0972,B 14.7767,C -0.1922,E1 14.6296,E2 292.3609} C_DIS
LIN {X -120.702,Y 46.5577,Z 158,A 158.5209,B 14.7767,C -0.1886,E1 14.6282,E2 290.9374} C_DIS
LIN {X -122.0846,Y 42.8023,Z 158,A 160.473,B 14.7767,C -0.1883,E1 14.6263,E2 288.967} C_DIS
LIN {X -123.3319,Y 39.0621,Z 158,A 162.0727,B 14.7769,C -0.1793,E1 14.625,E2 287.3864} C_DIS
LIN {X -124.2558,Y 36.0157,Z 158,A 163.5086,B 14.7769,C -0.1759,E1 14.6238,E2 285.9493} C_DIS
LIN {X -125.0984,Y 32.9704,Z 158,A 164.9094,B 14.7769,C -0.1718,E1 14.6228,E2 284.5502} C_DIS
LIN {X -125.8692,Y 29.894,Z 158,A 166.3275,B 14.7769,C -0.168,E1 14.6219,E2 283.1323} C_DIS
LIN {X -126.5663,Y 26.7914,Z 158,A 167.7485,B 14.777,C -0.1642,E1 14.621,E2 281.7118} C_DIS
LIN {X -127.1901,Y 23.6568,Z 158,A 169.1743,B 14.777,C -0.1603,E1 14.6203,E2 280.2866} C_DIS
LIN {X -127.7319,Y 20.535,Z 158,A 170.6159,B 14.7771,C -0.1571,E1 14.6196,E2 278.8424} C_DIS
LIN {X -128.1956,Y 17.4011,Z 158,A 172.0329,B 14.7771,C -0.1532,E1 14.619,E2 277.4256} C_DIS
LIN {X -128.5815,Y 14.2672,Z 158,A 173.4433,B 14.7771,C -0.1494,E1 14.6186,E2 276.0154} C_DIS
LIN {X -128.8929,Y 11.1012,Z 158,A 174.8632,B 14.7772,C -0.1454,E1 14.6182,E2 274.596} C_DIS
LIN {X -129.1369,Y 7.7639,Z 158,A 176.493,B 14.7772,C -0.1449,E1 14.6179,E2 272.9511} C_DIS
LIN {X -129.3341,Y 3.0911,Z 158,A 178.4296,B 14.7773,C -0.1351,E1 14.6177,E2 271.0326} C_DIS
LIN {X -129.3725,Y -0.0564,Z 158,A 179.8987,B 14.7773,C -0.1328,E1 14.6177,E2 269.5566} C_DIS
LIN {X -129.3312,Y -3.193,Z 158,A -178.5768,B 14.7773,C -0.1323,E1 14.6178,E2 268.0181} C_DIS
LIN {X -129.1268,Y -7.9284,Z 158,A -176.6162,B 14.7774,C -0.1223,E1 14.6181,E2 266.076} C_DIS
LIN {X -128.8938,Y -11.0916,Z 158,A -175.0886,B 14.7774,C -0.1214,E1 14.6184,E2 264.5358} C_DIS
LIN {X -128.5825,Y -14.2577,Z 158,A -173.7819,B 14.7774,C -0.1145,E1 14.6188,E2 263.2426} C_DIS
LIN {X -128.1292,Y -17.8783,Z 158,A -172.2851,B 14.7775,C -0.1065,E1 14.6194,E2 261.7614} C_DIS
LIN {X -127.7273,Y -20.5628,Z 158,A -170.9163,B 14.7775,C -0.1074,E1 14.6199,E2 260.3748} C_DIS
LIN {X -127.187,Y -23.6729,Z 158,A -169.4986,B 14.7775,C -0.1038,E1 14.6206,E2 258.9563} C_DIS
LIN {X -126.5661,Y -26.7924,Z 158,A -168.0752,B 14.7775,C -0.1001,E1 14.6214,E2 257.5328} C_DIS
LIN {X -125.8662,Y -29.9063,Z 158,A -166.6558,B 14.7776,C -0.0961,E1 14.6223,E2 256.1141} C_DIS
LIN {X -125.0945,Y -32.9849,Z 158,A -165.241,B 14.7776,C -0.0923,E1 14.6233,E2 254.6998} C_DIS
LIN {X -124.2488,Y -36.0396,Z 158,A -163.8182,B 14.7776,C -0.0888,E1 14.6244,E2 253.2763} C_DIS
LIN {X -123.2542,Y -39.3054,Z 158,A -162.3519,B 14.7776,C -0.0833,E1 14.6256,E2 251.8168} C_DIS
LIN {X -122.3321,Y -42.0884,Z 158,A -160.8555,B 14.7776,C -0.085,E1 14.627,E2 250.2987} C_DIS
LIN {X -121.2585,Y -45.0884,Z 158,A -159.5558,B 14.7777,C -0.078,E1 14.6282,E2 249.0133} C_DIS
LIN {X -120.1142,Y -48.0538,Z 158,A -158.1384,B 14.7777,C -0.0744,E1 14.6297,E2 247.5962} C_DIS
LIN {X -118.902,Y -50.9797,Z 158,A -156.7272,B 14.7777,C -0.0708,E1 14.6312,E2 246.1853} C_DIS
LIN {X -117.6239,Y -53.8638,Z 158,A -155.3152,B 14.7777,C -0.0675,E1 14.6328,E2 244.7728} C_DIS
LIN {X -116.2718,Y -56.7243,Z 158,A -153.7737,B 14.7777,C -0.0675,E1 14.6347,E2 243.2163} C_DIS
LIN {X -114.8344,Y -59.5812,Z 158,A -152.4857,B 14.7777,C -0.0604,E1 14.6363,E2 241.9445} C_DIS
LIN {X -113.3326,Y -62.3923,Z 158,A -151.0403,B 14.7778,C -0.0576,E1 14.6383,E2 240.4964} C_DIS
LIN {X -111.7683,Y -65.1535,Z 158,A -149.4663,B 14.7778,C -0.0587,E1 14.6405,E2 238.9038} C_DIS
LIN {X -110.1358,Y -67.8759,Z 158,A -148.1514,B 14.7778,C -0.0527,E1 14.6424,E2 237.6007} C_DIS
LIN {X -108.4433,Y -70.5481,Z 158,A -146.7906,B 14.7778,C -0.0481,E1 14.6444,E2 236.2456} C_DIS
LIN {X -106.687,Y -73.1768,Z 158,A -145.2278,B 14.7778,C -0.0492,E1 14.6469,E2 234.6648} C_DIS
LIN {X -104.8426,Y -75.7959,Z 158,A -143.9549,B 14.7778,C -0.0419,E1 14.649,E2 233.41} C_DIS
LIN {X -102.4737,Y -78.9698,Z 158,A -142.0209,B 14.7778,C -0.0427,E1 14.6522,E2 231.4561} C_DIS
LIN {X -99.4995,Y -82.6853,Z 158,A -140.051,B 14.7778,C -0.0342,E1 14.6557,E2 229.5037} C_DIS
LIN {X -96.9203,Y -85.6938,Z 158,A -138.1309,B 14.7778,C -0.0349,E1 14.6592,E2 227.5653} C_DIS
LIN {X -94.8495,Y -87.9807,Z 158,A -136.753,B 14.7778,C -0.0324,E1 14.6619,E2 226.1869} C_DIS
LIN {X -92.037,Y -90.9192,Z 158,A -135.0927,B 14.7778,C -0.0247,E1 14.6651,E2 224.5442} C_DIS
LIN {X -89.1959,Y -93.7076,Z 158,A -133.1577,B 14.7778,C -0.026,E1 14.669,E2 222.5899} C_DIS
LIN {X -85.6956,Y -96.9187,Z 158,A -131.0483,B 14.7779,C -0.0222,E1 14.6734,E2 220.4807} C_DIS
LIN {X -82.0858,Y -99.9948,Z 158,A -128.9405,B 14.7779,C -0.0186,E1 14.6779,E2 218.373} C_DIS
LIN {X -78.3422,Y -102.9542,Z 158,A -126.9546,B 14.7779,C -0.0113,E1 14.6822,E2 216.4029} C_DIS
LIN {X -75.7895,Y -104.8472,Z 158,A -125.5429,B 14.7779,C -0.0091,E1 14.6854,E2 214.9911} C_DIS
LIN {X -73.1938,Y -106.6754,Z 158,A -124.1099,B 14.7779,C -0.0076,E1 14.6887,E2 213.5554} C_DIS
LIN {X -70.5326,Y -108.4534,Z 158,A -122.7211,B 14.7779,C -0.0046,E1 14.6919,E2 212.1703} C_DIS
LIN {X -67.9045,Y -110.1183,Z 158,A -121.3091,B 14.7779,C -0.0036,E1 14.6953,E2 210.7546} C_DIS
LIN {X -65.1423,Y -111.7748,Z 158,A -119.8889,B 14.7779,C -0.0014,E1 14.6987,E2 209.3355} C_DIS
LIN {X -62.3811,Y -113.3388,Z 158,A -118.4706,B 14.7779,C 0.0001,E1 14.7021,E2 207.9159} C_DIS
LIN {X -59.5756,Y -114.8373,Z 158,A -117.0536,B 14.7779,C 0.0017,E1 14.7057,E2 206.498} C_DIS
LIN {X -56.7426,Y -116.2628,Z 158,A -115.6452,B 14.7779,C 0.0032,E1 14.7092,E2 205.0894} C_DIS
LIN {X -53.6915,Y -117.7036,Z 158,A -114.0023,B 14.7779,C 0.0006,E1 14.7134,E2 203.429} C_DIS
LIN {X -49.504,Y -119.5239,Z 158,A -112.1186,B 14.7779,C 0.0067,E1 14.7182,E2 201.5617} C_DIS
LIN {X -46.5492,Y -120.7053,Z 158,A -110.5626,B 14.7779,C 0.0038,E1 14.7223,E2 199.9884} C_DIS
LIN {X -41.9284,Y -122.3876,Z 158,A -108.5366,B 14.7779,C 0.0102,E1 14.7276,E2 197.9803} C_DIS
LIN {X -39.0628,Y -123.3317,Z 158,A -107.1829,B 14.7779,C 0.0107,E1 14.7312,E2 196.6243} C_DIS
LIN {X -35.5069,Y -124.4036,Z 158,A -105.5484,B 14.7779,C 0.0122,E1 14.7355,E2 194.9909} C_DIS
LIN {X -32.9776,Y -125.0965,Z 158,A -104.3719,B 14.7779,C 0.0124,E1 14.7387,E2 193.8124} C_DIS
LIN {X -29.9055,Y -125.8664,Z 158,A -102.9682,B 14.7779,C 0.0132,E1 14.7425,E2 192.4083} C_DIS
LIN {X -26.8178,Y -126.5606,Z 158,A -101.5651,B 14.7779,C 0.0138,E1 14.7464,E2 191.0048} C_DIS
LIN {X -23.1237,Y -127.2869,Z 158,A -100.0696,B 14.7779,C 0.0196,E1 14.7504,E2 189.5292} C_DIS
LIN {X -20.1829,Y -127.7864,Z 158,A -98.6872,B 14.7779,C 0.0183,E1 14.7542,E2 188.1392} C_DIS
LIN {X -17.3981,Y -128.196,Z 158,A -97.3075,B 14.7779,C 0.0147,E1 14.7581,E2 186.7434} C_DIS
LIN {X -14.2599,Y -128.5823,Z 158,A -95.9094,B 14.7779,C 0.015,E1 14.762,E2 185.3451} C_DIS
LIN {X -11.0349,Y -128.8985,Z 158,A -94.4897,B 14.7779,C 0.0156,E1 14.7659,E2 183.9266} C_DIS
LIN {X -7.9166,Y -129.1275,Z 158,A -93.1023,B 14.7779,C 0.0156,E1 14.7698,E2 182.5383} C_DIS
LIN {X -4.7503,Y -129.2831,Z 158,A -91.7054,B 14.7779,C 0.0158,E1 14.7737,E2 181.1417} C_DIS
LIN {X -1.5911,Y -129.3615,Z 158,A -90.3143,B 14.7779,C 0.0159,E1 14.7776,E2 179.7509} C_DIS
LIN {X 0.9078,Y -129.3647,Z 158,A -89.4432,B 14.7779,C 0.0228,E1 14.7799,E2 178.9071} C_DIS
Enddeposition()
LIN {X 0.9597,Y -137.0527,Z 159,A -92.8598,B 24.9713,C -1.2377,E1 25.0005,E2 179.5674} C_DIS
Startdeposition()
$VEL.CP = VEL_PRINT
LIN {X -5.2813,Y -136.9557,Z 159,A -95.4325,B 24.9713,C -1.2392,E1 24.9934,E2 182.1367} C_DIS
LIN {X -8.4201,Y -136.7985,Z 159,A -96.84,B 24.9715,C -1.2341,E1 24.9894,E2 183.5568} C_DIS
LIN {X -12.4091,Y -136.4962,Z 159,A -99.1922,B 24.9731,C -1.1978,E1 24.9826,E2 185.9961} C_DIS
LIN {X -17.8456,Y -135.8905,Z 159,A -100.435,B 24.9705,C -1.2541,E1 24.9795,E2 187.1064} C_DIS
LIN {X -24.6121,Y -134.8301,Z 159,A -103.6254,B 24.9713,C -1.2373,E1 24.9706,E2 190.3395} C_DIS
LIN {X -28.0212,Y -134.164,Z 159,A -105.2172,B 24.9716,C -1.2305,E1 24.9662,E2 191.9494} C_DIS
LIN {X -31.9677,Y -133.277,Z 159,A -106.7877,B 24.9713,C -1.2378,E1 24.962,E2 193.5045} C_DIS
LIN {X -35.4042,Y -132.4055,Z 159,A -108.2494,B 24.9713,C -1.2398,E1 24.958,E2 194.9637} C_DIS
LIN {X -38.6063,Y -131.5074,Z 159,A -109.6605,B 24.9713,C -1.2396,E1 24.9542,E2 196.3774} C_DIS
LIN {X -42.0011,Y -130.4632,Z 159,A -111.1444,B 24.9712,C -1.2408,E1 24.9503,E2 197.8611} C_DIS
LIN {X -45.5688,Y -129.2618,Z 159,A -112.7992,B 24.9713,C -1.2379,E1 24.9459,E2 199.5261} C_DIS
LIN {X -50.174,Y -127.5441,Z 159,A -114.7347,B 24.9709,C -1.2462,E1 24.9409,E2 201.446} C_DIS
LIN {X -59.4901,Y -123.4736,Z 159,A -119.0248,B 24.9708,C -1.2488,E1 24.93,E2 205.7402} C_DIS
LIN {X -62.411,Y -122.0226,Z 159,A -120.435,B 24.9708,C -1.2481,E1 24.9264,E2 207.1557} C_DIS
LIN {X -65.7883,Y -120.2375,Z 159,A -122.0656,B 24.9708,C -1.2485,E1 24.9224,E2 208.79} C_DIS
LIN {X -69.2875,Y -118.2556,Z 159,A -123.7412,B 24.9707,C -1.2512,E1 24.9183,E2 210.4641} C_DIS
LIN {X -72.9712,Y -116.0189,Z 159,A -125.5168,B 24.9705,C -1.2554,E1 24.9141,E2 212.2355} C_DIS
LIN {X -76.4632,Y -113.7484,Z 159,A -127.3783,B 24.9706,C -1.252,E1 24.9097,E2 214.1111} C_DIS
LIN {X -80.238,Y -111.1173,Z 159,A -129.2867,B 24.9705,C -1.2561,E1 24.9054,E2 216.0163} C_DIS
LIN {X -84.576,Y -107.8519,Z 159,A -132.8635,B 24.9733,C -1.1937,E1 24.8972,E2 219.7546} C_DIS
LIN {X -91.6689,Y -101.8923,Z 159,A -135.4422,B 24.9699,C -1.2672,E1 24.8921,E2 222.1686} C_DIS
LIN {X -94.8396,Y -98.9476,Z 159,A -137.1658,B 24.9695,C -1.2754,E1 24.8886,E2 223.8799} C_DIS
LIN {X -98.0521,Y -95.7654,Z 159,A -139.0618,B 24.9694,C -1.2792,E1 24.8849,E2 225.7747} C_DIS
LIN {X -100.7847,Y -92.8849,Z 159,A -140.8347,B 24.9694,C -1.2772,E1 24.8815,E2 227.5602} C_DIS
LIN {X -104.6024,Y -88.5637,Z 159,A -143.0012,B 24.9686,C -1.2954,E1 24.8776,E2 229.6933} C_DIS
LIN {X -106.6129,Y -86.1326,Z 159,A -144.5766,B 24.9691,C -1.2854,E1 24.8747,E2 231.2996} C_DIS
LIN {X -109.3879,Y -82.5798,Z 159,A -146.4465,B 24.9688,C -1.2909,E1 24.8716,E2 233.1655} C_DIS
LIN {X -112.0394,Y -78.945,Z 159,A -148.3045,B 24.9685,C -1.2969,E1 24.8685,E2 235.0183} C_DIS
LIN {X -114.6324,Y -75.1307,Z 159,A -150.3828,B 24.9686,C -1.2943,E1 24.8653,E2 237.113} C_DIS
LIN {X -117.294,Y -70.9031,Z 159,A -152.3941,B 24.9682,C -1.3039,E1 24.8624,E2 239.1119} C_DIS
LIN {X -119.6031,Y -66.935,Z 159,A -154.4055,B 24.9682,C -1.3045,E1 24.8596,E2 241.1321} C_DIS
LIN {X -121.9446,Y -62.5643,Z 159,A -156.3712,B 24.9676,C -1.3158,E1 24.857,E2 243.0814} C_DIS
LIN {X -125.3825,Y -55.3559,Z 159,A -159.6379,B 24.9669,C -1.3291,E1 24.8532,E2 246.3343} C_DIS
LIN {X -126.5013,Y -52.7449,Z 159,A -160.8574,B 24.9669,C -1.3311,E1 24.8518,E2 247.5559} C_DIS
LIN {X -127.8352,Y -49.4252,Z 159,A -162.3667,B 24.9666,C -1.3349,E1 24.8503,E2 249.0646} C_DIS
LIN {X -128.9927,Y -46.32,Z 159,A -163.7782,B 24.9665,C -1.3378,E1 24.8489,E2 250.4772} C_DIS
LIN {X -130.1383,Y -42.9971,Z 159,A -165.3409,B 24.9665,C -1.3376,E1 24.8475,E2 252.0492} C_DIS
LIN {X -132.2984,Y -35.8057,Z 159,A -168.2815,B 24.9655,C -1.3573,E1 24.8452,E2 254.9598} C_DIS
LIN {X -133.3901,Y -31.4984,Z 159,A -170.2549,B 24.9655,C -1.3573,E1 24.8439,E2 256.9447} C_DIS
LIN {X -134.1332,Y -28.1701,Z 159,A -172.0299,B 24.9661,C -1.3445,E1 24.8428,E2 258.7608} C_DIS
LIN {X -134.7854,Y -24.8619,Z 159,A -173.0881,B 24.965,C -1.3665,E1 24.8423,E2 259.7727} C_DIS
LIN {X -135.4796,Y -20.737,Z 159,A -174.9089,B 24.965,C -1.3686,E1 24.8415,E2 261.5994} C_DIS
LIN {X -135.9431,Y -17.4444,Z 159,A -176.2572,B 24.9646,C -1.3752,E1 24.841,E2 262.9401} C_DIS
LIN {X -136.2901,Y -14.4829,Z 159,A -177.55,B 24.9645,C -1.377,E1 24.8406,E2 264.2363} C_DIS
LIN {X -136.6692,Y -10.3141,Z 159,A -179.3369,B 24.9643,C -1.3809,E1 24.8402,E2 266.0247} C_DIS
LIN {X -136.8931,Y -6.7108,Z 159,A 179.119,B 24.9641,C -1.3841,E1 24.8399,E2 267.5703} C_DIS
LIN {X -137.0364,Y -2.4086,Z 159,A 177.3632,B 24.9637,C -1.3922,E1 24.8398,E2 269.3174} C_DIS
LIN {X -137.0505,Y 1.5615,Z 159,A 175.5605,B 24.9637,C -1.3906,E1 24.8398,E2 271.1349} C_DIS
LIN {X -136.9532,Y 5.3435,Z 159,A 174.0686,B 24.9633,C -1.4003,E1 24.84,E2 272.6125} C_DIS
LIN {X -136.7414,Y 9.3239,Z 159,A 172.2888,B 24.9633,C -1.4003,E1 24.8403,E2 274.4034} C_DIS
LIN {X -136.4217,Y 13.1852,Z 159,A 170.8046,B 24.9626,C -1.4123,E1 24.8406,E2 275.8676} C_DIS
LIN {X -136.055,Y 16.5484,Z 159,A 169.3535,B 24.9625,C -1.4152,E1 24.8411,E2 277.3205} C_DIS
LIN {X -135.5921,Y 19.9966,Z 159,A 167.7709,B 24.9625,C -1.4136,E1 24.8417,E2 278.9163} C_DIS
LIN {X -134.9142,Y 24.1423,Z 159,A 166.1318,B 24.9619,C -1.4253,E1 24.8425,E2 280.5374} C_DIS
LIN {X -134.2508,Y 27.5945,Z 159,A 164.5724,B 24.9619,C -1.4256,E1 24.8433,E2 282.1051} C_DIS
LIN {X -133.3182,Y 31.7965,Z 159,A 162.7708,B 24.9616,C -1.4314,E1 24.8444,E2 283.9035} C_DIS
LIN {X -132.3424,Y 35.6407,Z 159,A 161.1395,B 24.9613,C -1.4382,E1 24.8456,E2 285.5282} C_DIS
LIN {X -131.4344,Y 38.8559,Z 159,A 159.727,B 24.9611,C -1.4419,E1 24.8467,E2 286.9401} C_DIS
LIN {X -130.3621,Y 42.3176,Z 159,A 157.9904,B 24.9614,C -1.4357,E1 24.8482,E2 288.7013} C_DIS
LIN {X -128.882,Y 46.6268,Z 159,A 156.2829,B 24.9605,C -1.4516,E1 24.8497,E2 290.3806} C_DIS
LIN {X -127.5872,Y 50.063,Z 159,A 154.7846,B 24.9602,C -1.4583,E1 24.8512,E2 291.8713} C_DIS
LIN {X -126.3572,Y 53.0901,Z 159,A 153.3766,B 24.96,C -1.4605,E1 24.8527,E2 293.2819} C_DIS
LIN {X -124.9387,Y 56.348,Z 159,A 151.8759,B 24.9598,C -1.4644,E1 24.8544,E2 294.7817} C_DIS
LIN {X -123.518,Y 59.3971,Z 159,A 150.4822,B 24.9596,C -1.4694,E1 24.8561,E2 296.1711} C_DIS
LIN {X -121.8535,Y 62.7431,Z 159,A 148.8811,B 24.9594,C -1.4722,E1 24.8581,E2 297.7741} C_DIS
LIN {X -119.8103,Y 66.5632,Z 159,A 146.9753,B 24.9594,C -1.4729,E1 24.8607,E2 299.6883} C_DIS
LIN {X -117.4615,Y 70.6262,Z 159,A 145.0759,B 24.9589,C -1.4818,E1 24.8633,E2 301.5763} C_DIS
LIN {X -114.2567,Y 75.7014,Z 159,A 142.6587,B 24.9582,C -1.4937,E1 24.867,E2 303.9775} C_DIS
LIN {X -109.4955,Y 82.4372,Z 159,A 138.9983,B 24.9582,C -1.4927,E1 24.873,E2 307.6581} C_DIS
LIN {X -106.75,Y 85.9626,Z 159,A 137.18,B 24.9578,C -1.5002,E1 24.8761,E2 309.4669} C_DIS
LIN {X -104.1974,Y 89.0401,Z 159,A 135.5002,B 24.9576,C -1.5043,E1 24.8791,E2 311.1449} C_DIS
LIN {X -100.9364,Y 92.7199,Z 159,A 133.4222,B 24.9574,C -1.5085,E1 24.883,E2 313.2221} C_DIS
LIN {X -98.0589,Y 95.7584,Z 159,A 131.6477,B 24.9572,C -1.5116,E1 24.8864,E2 314.9968} C_DIS
LIN {X -95.0498,Y 98.7462,Z 159,A 129.8287,B 24.9571,C -1.5137,E1 24.89,E2 316.8186} C_DIS
LIN {X -91.595,Y 101.9585,Z 159,A 127.8957,B 24.9567,C -1.5203,E1 24.894,E2 318.7435} C_DIS
LIN {X -88.4865,Y 104.6681,Z 159,A 126.1693,B 24.9565,C -1.5242,E1 24.8977,E2 320.4675} C_DIS
LIN {X -85.2321,Y 107.3343,Z 159,A 124.4061,B 24.9563,C -1.5279,E1 24.9015,E2 322.2284} C_DIS
LIN {X -82.0617,Y 109.7774,Z 159,A 122.6531,B 24.9563,C -1.5275,E1 24.9054,E2 323.9888} C_DIS
LIN {X -78.2067,Y 112.556,Z 159,A 120.7386,B 24.9558,C -1.5353,E1 24.9097,E2 325.8913} C_DIS
LIN {X -74.7182,Y 114.9014,Z 159,A 118.9395,B 24.9558,C -1.5366,E1 24.9139,E2 327.6931} C_DIS
LIN {X -69.0041,Y 118.4218,Z 159,A 116.0979,B 24.9556,C -1.5401,E1 24.9207,E2 330.5352} C_DIS
LIN {X -65.1461,Y 120.587,Z 159,A 114.2296,B 24.9554,C -1.5424,E1 24.9253,E2 332.4035} C_DIS
LIN {X -61.7722,Y 122.3478,Z 159,A 112.7663,B 24.9549,C -1.5516,E1 24.9289,E2 333.8487} C_DIS
LIN {X -58.6822,Y 123.8595,Z 159,A 111.2958,B 24.9549,C -1.5523,E1 24.9326,E2 335.3214} C_DIS
LIN {X -55.4452,Y 125.3425,Z 159,A 109.8415,B 24.9546,C -1.5563,E1 24.9363,E2 336.7697} C_DIS
LIN {X -52.5195,Y 126.5955,Z 159,A 108.436,B 24.9547,C -1.5544,E1 24.9399,E2 338.1829} C_DIS
LIN {X -47.5016,Y 128.5636,Z 159,A 106.3006,B 24.9542,C -1.5636,E1 24.9454,E2 340.301} C_DIS
LIN {X -44.9969,Y 129.4601,Z 159,A 104.7724,B 24.9554,C -1.5436,E1 24.9496,E2 341.8798} C_DIS
LIN {X -41.6411,Y 130.5782,Z 159,A 103.9012,B 24.9534,C -1.5768,E1 24.9517,E2 342.6737} C_DIS
LIN {X -36.0084,Y 132.2443,Z 159,A 101.2199,B 24.954,C -1.5677,E1 24.959,E2 345.381} C_DIS
LIN {X -31.5209,Y 133.3846,Z 159,A 99.2513,B 24.954,C -1.5679,E1 24.9643,E2 347.3519} C_DIS
LIN {X -28.5061,Y 134.0606,Z 159,A 97.9636,B 24.9539,C -1.5693,E1 24.9678,E2 348.6379} C_DIS
LIN {X -25.4189,Y 134.6798,Z 159,A 96.6209,B 24.9539,C -1.569,E1 24.9715,E2 349.9828} C_DIS
LIN {X -21.4127,Y 135.375,Z 159,A 94.8609,B 24.9539,C -1.5671,E1 24.9764,E2 351.7489} C_DIS
LIN {X -17.4921,Y 135.9369,Z 159,A 93.2702,B 24.9537,C -1.5716,E1 24.9807,E2 353.3303} C_DIS
LIN {X -13.4581,Y 136.3955,Z 159,A 91.493,B 24.9539,C -1.5683,E1 24.9857,E2 355.1163} C_DIS
LIN {X -9.8924,Y 136.6999,Z 159,A 90.0864,B 24.9536,C -1.5737,E1 24.9896,E2 356.5107} C_DIS
LIN {X -6.618,Y 136.8978,Z 159,A 88.6037,B 24.9539,C -1.5683,E1 24.9937,E2 358.0066} C_DIS
LIN {X 0.5803,Y 137.0564,Z 159,A 85.7904,B 24.9533,C -1.5795,E1 25.0015,E2 360.7936} C_DIS
LIN {X 3.0538,Y 137.0255,Z 159,A 84.453,B 24.9542,C -1.5635,E1 25.0054,E2 362.1686} C_DIS
LIN {X 7.9493,Y 136.8275,Z 159,A 82.5251,B 24.9538,C -1.57,E1 25.0107,E2 364.0806} C_DIS
LIN {X 13.7945,Y 136.3632,Z 159,A 80.2568,B 24.9533,C -1.5795,E1 25.017,E2 366.3251} C_DIS
LIN {X 18.1845,Y 135.8461,Z 159,A 78.1721,B 24.954,C -1.5665,E1 25.0228,E2 368.439} C_DIS
LIN {X 22.403,Y 135.214,Z 159,A 76.5059,B 24.9537,C -1.5722,E1 25.0274,E2 370.0901} C_DIS
LIN {X 26.0671,Y 134.5559,Z 159,A 74.9812,B 24.9537,C -1.5732,E1 25.0315,E2 371.6106} C_DIS
LIN {X 29.2393,Y 133.9023,Z 159,A 73.6294,B 24.9537,C -1.5726,E1 25.0352,E2 372.962} C_DIS
LIN {X 32.797,Y 133.0771,Z 159,A 71.9501,B 24.9542,C -1.5635,E1 25.0398,E2 374.6605} C_DIS
LIN {X 36.7726,Y 132.032,Z 159,A 70.3269,B 24.954,C -1.5675,E1 25.0442,E2 376.2716} C_DIS
LIN {X 40.3446,Y 130.9848,Z 159,A 68.778,B 24.954,C -1.5667,E1 25.0483,E2 377.8198} C_DIS
LIN {X 44.2404,Y 129.7224,Z 159,A 66.9189,B 24.9546,C -1.5573,E1 25.0533,E2 379.6977} C_DIS
LIN {X 48.2301,Y 128.2907,Z 159,A 65.3275,B 24.9541,C -1.5654,E1 25.0574,E2 381.2666} C_DIS
LIN {X 56.3547,Y 124.9357,Z 159,A 61.6848,B 24.9542,C -1.563,E1 25.0668,E2 384.9063} C_DIS
LIN {X 59.3594,Y 123.536,Z 159,A 60.2613,B 24.9544,C -1.5592,E1 25.0704,E2 386.3351} C_DIS
LIN {X 62.5357,Y 121.9591,Z 159,A 58.7416,B 24.9547,C -1.5552,E1 25.0742,E2 387.86} C_DIS
LIN {X 66.3652,Y 119.9199,Z 159,A 56.9227,B 24.9548,C -1.5524,E1 25.0787,E2 389.6804} C_DIS
LIN {X 70.2044,Y 117.7136,Z 159,A 55.2423,B 24.9545,C -1.559,E1 25.0827,E2 391.3401} C_DIS
LIN {X 73.384,Y 115.7584,Z 159,A 53.5044,B 24.9552,C -1.5467,E1 25.0868,E2 393.1014} C_DIS
LIN {X 76.8769,Y 113.4684,Z 159,A 51.7555,B 24.9554,C -1.5437,E1 25.0909,E2 394.8518} C_DIS
LIN {X 80.5196,Y 110.9132,Z 159,A 50.0524,B 24.955,C -1.549,E1 25.0947,E2 396.5362} C_DIS
LIN {X 83.3578,Y 108.7962,Z 159,A 48.4506,B 24.9556,C -1.5396,E1 25.0983,E2 398.1546} C_DIS
LIN {X 86.8663,Y 106.0161,Z 159,A 46.3043,B 24.9567,C -1.5208,E1 25.1031,E2 400.337} C_DIS
LIN {X 89.6798,Y 103.6473,Z 159,A 45.032,B 24.956,C -1.5324,E1 25.1057,E2 401.5771} C_DIS
LIN {X 92.9895,Y 100.6886,Z 159,A 43.2409,B 24.956,C -1.5321,E1 25.1094,E2 403.3617} C_DIS
LIN {X 96.0883,Y 97.7353,Z 159,A 41.5069,B 24.956,C -1.5313,E1 25.1129,E2 405.0903} C_DIS
LIN {X 98.7741,Y 95.021,Z 159,A 39.8241,B 24.9565,C -1.5229,E1 25.1162,E2 406.7857} C_DIS
LIN {X 101.4936,Y 92.1096,Z 159,A 38.2002,B 24.9566,C -1.5214,E1 25.1192,E2 408.406} C_DIS
LIN {X 104.3531,Y 88.857,Z 159,A 36.3526,B 24.957,C -1.515,E1 25.1226,E2 410.2603} C_DIS
LIN {X 107.315,Y 85.2563,Z 159,A 34.421,B 24.9572,C -1.5112,E1 25.126,E2 412.1919} C_DIS
LIN {X 109.8945,Y 81.9044,Z 159,A 32.6985,B 24.9573,C -1.5093,E1 25.1289,E2 413.9107} C_DIS
LIN {X 112.375,Y 78.4668,Z 159,A 30.589,B 24.9586,C -1.4859,E1 25.1324,E2 416.0653} C_DIS
LIN {X 114.5666,Y 75.2307,Z 159,A 29.5242,B 24.9571,C -1.5134,E1 25.1339,E2 417.0597} C_DIS
LIN {X 116.2684,Y 72.5728,Z 159,A 27.9667,B 24.958,C -1.4965,E1 25.1363,E2 418.6494} C_DIS
LIN {X 118.5928,Y 68.7087,Z 159,A 26.1303,B 24.9582,C -1.494,E1 25.1389,E2 420.4821} C_DIS
LIN {X 120.5757,Y 65.1672,Z 159,A 24.4695,B 24.9583,C -1.4913,E1 25.1411,E2 422.1407} C_DIS
LIN {X 122.191,Y 62.0803,Z 159,A 23.0953,B 24.9583,C -1.4918,E1 25.1429,E2 423.5064} C_DIS
LIN {X 123.9454,Y 58.5026,Z 159,A 21.3909,B 24.9587,C -1.4848,E1 25.145,E2 425.2182} C_DIS
LIN {X 125.339,Y 55.4531,Z 159,A 20.0027,B 24.9589,C -1.4814,E1 25.1466,E2 426.6068} C_DIS
LIN {X 126.6016,Y 52.5048,Z 159,A 18.6675,B 24.9591,C -1.4777,E1 25.148,E2 427.9434} C_DIS
LIN {X 128.1313,Y 48.6557,Z 159,A 16.1251,B 24.9619,C -1.4268,E1 25.1507,E2 430.5917} C_DIS
LIN {X 130.1841,Y 42.8595,Z 159,A 14.669,B 24.9589,C -1.4818,E1 25.1519,E2 431.9098} C_DIS
LIN {X 130.9798,Y 40.3608,Z 159,A 13.244,B 24.9601,C -1.4597,E1 25.1531,E2 433.3789} C_DIS
LIN {X 132.0082,Y 36.8577,Z 159,A 11.8097,B 24.9601,C -1.4601,E1 25.1542,E2 434.804} C_DIS
LIN {X 132.9107,Y 33.4584,Z 159,A 10.3529,B 24.9603,C -1.4563,E1 25.1552,E2 436.2615} C_DIS
LIN {X 133.6395,Y 30.4165,Z 159,A 9.0118,B 24.9606,C -1.4502,E1 25.156,E2 437.6091} C_DIS
LIN {X 134.502,Y 26.3493,Z 159,A 7.2142,B 24.9611,C -1.4412,E1 25.157,E2 439.4175} C_DIS
LIN {X 135.1779,Y 22.6189,Z 159,A 5.7122,B 24.9611,C -1.4408,E1 25.1578,E2 440.9115} C_DIS
LIN {X 135.7591,Y 18.8275,Z 159,A 4.154,B 24.9613,C -1.4382,E1 25.1584,E2 442.4669} C_DIS
LIN {X 136.2428,Y 14.9225,Z 159,A 2.4408,B 24.9618,C -1.4289,E1 25.159,E2 444.1918} C_DIS
LIN {X 136.6474,Y 10.6125,Z 159,A 0.119,B 24.9636,C -1.3938,E1 25.1595,E2 446.5824} C_DIS
LIN {X 136.9363,Y 5.7751,Z 159,A -1.2823,B 24.9621,C -1.4226,E1 25.1597,E2 447.9075} C_DIS
LIN {X 137.0477,Y 1.7289,Z 159,A -3.5301,B 24.9641,C -1.3853,E1 25.1597,E2 450.2298} C_DIS
LIN {X 137.0272,Y -2.9467,Z 159,A -5.4164,B 24.9641,C -1.3827,E1 25.1597,E2 452.111} C_DIS
LIN {X 136.8666,Y -7.2388,Z 159,A -6.7356,B 24.9631,C -1.4039,E1 25.1595,E2 453.3726} C_DIS
LIN {X 136.5824,Y -11.4017,Z 159,A -8.4651,B 24.9633,C -1.3989,E1 25.1591,E2 455.1035} C_DIS
LIN {X 136.0938,Y -16.2228,Z 159,A -10.4596,B 24.9636,C -1.394,E1 25.1586,E2 457.0978} C_DIS
LIN {X 135.5072,Y -20.5587,Z 159,A -12.1113,B 24.9634,C -1.3981,E1 25.1579,E2 458.7301} C_DIS
LIN {X 134.8465,Y -24.5203,Z 159,A -13.9274,B 24.9641,C -1.3846,E1 25.1571,E2 460.5672} C_DIS
LIN {X 134.2159,Y -27.7664,Z 159,A -15.4405,B 24.9647,C -1.3726,E1 25.1562,E2 462.0999} C_DIS
LIN {X 133.2291,Y -32.1663,Z 159,A -17.1539,B 24.9645,C -1.3762,E1 25.1551,E2 463.7948} C_DIS
LIN {X 132.4573,Y -35.2096,Z 159,A -18.4853,B 24.9648,C -1.3708,E1 25.1542,E2 465.1312} C_DIS
LIN {X 131.5177,Y -38.5712,Z 159,A -19.9525,B 24.9651,C -1.3656,E1 25.1531,E2 466.6023} C_DIS
LIN {X 130.3877,Y -42.2372,Z 159,A -21.5182,B 24.9652,C -1.3626,E1 25.1518,E2 468.1663} C_DIS
LIN {X 129.3311,Y -45.3691,Z 159,A -22.8959,B 24.9654,C -1.3584,E1 25.1505,E2 469.5461} C_DIS
LIN {X 128.1834,Y -48.5166,Z 159,A -24.3002,B 24.9657,C -1.3537,E1 25.1491,E2 470.9535} C_DIS
LIN {X 126.8123,Y -51.9992,Z 159,A -26.2314,B 24.967,C -1.3278,E1 25.1471,E2 472.9351} C_DIS
LIN {X 125.359,Y -55.4084,Z 159,A -27.2956,B 24.9658,C -1.3506,E1 25.146,E2 473.9397} C_DIS
LIN {X 124.2066,Y -57.9442,Z 159,A -28.5647,B 24.9663,C -1.341,E1 25.1444,E2 475.2246} C_DIS
LIN {X 122.6807,Y -61.109,Z 159,A -30.0126,B 24.9665,C -1.3377,E1 25.1427,E2 476.6726} C_DIS
LIN {X 120.1765,Y -65.9002,Z 159,A -32.0995,B 24.9663,C -1.3407,E1 25.14,E2 478.7414} C_DIS
LIN {X 115.437,Y -73.888,Z 159,A -36.0069,B 24.967,C -1.3276,E1 25.1344,E2 482.6596} C_DIS
LIN {X 113.5679,Y -76.7298,Z 159,A -37.6101,B 24.9677,C -1.3132,E1 25.1318,E2 484.2889} C_DIS
LIN {X 111.0575,Y -80.3205,Z 159,A -39.3793,B 24.9677,C -1.3115,E1 25.129,E2 486.0534} C_DIS
LIN {X 108.5876,Y -83.6297,Z 159,A -41.4586,B 24.969,C -1.2867,E1 25.1254,E2 488.1814} C_DIS
LIN {X 106.1877,Y -86.6563,Z 159,A -42.643,B 24.968,C -1.3066,E1 25.1234,E2 489.3131} C_DIS
LIN {X 103.6526,Y -89.6736,Z 159,A -44.406,B 24.9686,C -1.2957,E1 25.1202,E2 491.094} C_DIS
LIN {X 100.9465,Y -92.7089,Z 159,A -46.041,B 24.9686,C -1.2949,E1 25.1171,E2 492.7236} C_DIS
LIN {X 97.3901,Y -96.4383,Z 159,A -48.0966,B 24.9686,C -1.2949,E1 25.1131,E2 494.7702} C_DIS
LIN {X 94.6016,Y -99.175,Z 159,A -49.8105,B 24.969,C -1.2864,E1 25.1097,E2 496.4972} C_DIS
LIN {X 91.5945,Y -101.9589,Z 159,A -51.5807,B 24.9694,C -1.279,E1 25.106,E2 498.2776} C_DIS
LIN {X 87.6515,Y -105.3681,Z 159,A -53.6031,B 24.9692,C -1.2828,E1 25.1017,E2 500.2832} C_DIS
LIN {X 84.6832,Y -107.7678,Z 159,A -55.3314,B 24.9697,C -1.2717,E1 25.0979,E2 502.0312} C_DIS
LIN {X 81.7595,Y -110.0024,Z 159,A -57.362,B 24.9712,C -1.2408,E1 25.0932,E2 504.1273} C_DIS
LIN {X 77.6856,Y -112.9164,Z 159,A -58.9041,B 24.9699,C -1.2673,E1 25.0899,E2 505.6018} C_DIS
LIN {X 74.1726,Y -115.2548,Z 159,A -60.6963,B 24.9702,C -1.2621,E1 25.0857,E2 507.4003} C_DIS
LIN {X 70.3957,Y -117.5995,Z 159,A -62.7144,B 24.9708,C -1.2496,E1 25.0808,E2 509.4415} C_DIS
LIN {X 66.8822,Y -119.6328,Z 159,A -64.2031,B 24.9704,C -1.2581,E1 25.0772,E2 510.9058} C_DIS
LIN {X 63.0035,Y -121.7201,Z 159,A -66.0612,B 24.9706,C -1.2539,E1 25.0726,E2 512.7685} C_DIS
LIN {X 56.5751,Y -124.8371,Z 159,A -68.8803,B 24.9703,C -1.2584,E1 25.0656,E2 515.5698} C_DIS
LIN {X 52.564,Y -126.5769,Z 159,A -70.7808,B 24.9707,C -1.2516,E1 25.0607,E2 517.4819} C_DIS
LIN {X 49.4176,Y -127.8381,Z 159,A -72.2065,B 24.9707,C -1.2491,E1 25.0569,E2 518.9103} C_DIS
LIN {X 45.782,Y -129.1867,Z 159,A -73.7856,B 24.9707,C -1.2491,E1 25.0528,E2 520.4859} C_DIS
LIN {X 42.6632,Y -130.2495,Z 159,A -75.1461,B 24.9708,C -1.2483,E1 25.0492,E2 521.8457} C_DIS
LIN {X 39.5427,Y -131.2302,Z 159,A -76.6782,B 24.9713,C -1.2376,E1 25.0451,E2 523.4004} C_DIS
LIN {X 34.2113,Y -132.7196,Z 159,A -78.7181,B 24.9707,C -1.2502,E1 25.0397,E2 525.4073} C_DIS
LIN {X 29.3988,Y -133.8679,Z 159,A -81.0074,B 24.9714,C -1.236,E1 25.0333,E2 527.727} C_DIS
LIN {X 25.6646,Y -134.6329,Z 159,A -82.4776,B 24.9711,C -1.2414,E1 25.0294,E2 529.1826} C_DIS
LIN {X 22.3721,Y -135.2191,Z 159,A -83.9177,B 24.9713,C -1.238,E1 25.0254,E2 530.6293} C_DIS
LIN {X 18.7568,Y -135.7692,Z 159,A -85.7099,B 24.972,C -1.2225,E1 25.0203,E2 532.4566} C_DIS
LIN {X 15.5229,Y -136.1768,Z 159,A -86.7158,B 24.9712,C -1.2411,E1 25.0177,E2 533.4178} C_DIS
LIN {X 7.7901,Y -136.8373,Z 159,A -90.9073,B 24.9736,C -1.1884,E1 25.0057,E2 537.7321} C_DIS
LIN {X 1.3309,Y -137.0522,Z 159,A -92.839,B 24.9717,C -1.2289,E1 25.0005,E2 539.5674} C_DIS
LIN {X 1.3309,Y -137.0522,Z 159,A -92.839,B 24.9717,C -1.2289,E1 25.0005,E2 539.5674} C_DIS
Enddeposition()
LIN {X 0.9413,Y -136.1203,Z 159,A -91.5841,B 23.9214,C -1.1033,E1 23.9489,E2 538.4853} C_DIS
Startdeposition()
$VEL.CP = VEL_PRINT
LIN {X 4.8969,Y -136.042,Z 159,A -90.2091,B 23.9221,C -1.0885,E1 23.9526,E2 537.1471} C_DIS
LIN {X 9.1898,Y -135.8208,Z 159,A -87.9324,B 23.921,C -1.1138,E1 23.9591,E2 534.8089} C_DIS
LIN {X 13.6137,Y -135.4483,Z 159,A -86.5728,B 23.9221,C -1.088,E1 23.9627,E2 533.5138} C_DIS
LIN {X 17.9635,Y -134.9392,Z 159,A -84.6973,B 23.9219,C -1.0909,E1 23.9679,E2 531.6328} C_DIS
LIN {X 22.1801,Y -134.3104,Z 159,A -82.9355,B 23.9219,C -1.0905,E1 23.9728,E2 529.8738} C_DIS
LIN {X 25.7276,Y -133.6761,Z 159,A -81.417,B 23.9219,C -1.0918,E1 23.977,E2 528.3538} C_DIS
LIN {X 29.9321,Y -132.7983,Z 159,A -79.5969,B 23.9219,C -1.0941,E1 23.9819,E2 526.5306} C_DIS
LIN {X 33.9946,Y -131.8172,Z 159,A -77.7113,B 23.9214,C -1.1026,E1 23.9871,E2 524.627} C_DIS
LIN {X 39.252,Y -130.3487,Z 159,A -75.4994,B 23.9215,C -1.1006,E1 23.993,E2 522.4238} C_DIS
LIN {X 42.6731,Y -129.2681,Z 159,A -74.0566,B 23.9216,C -1.0989,E1 23.9968,E2 520.9881} C_DIS
LIN {X 46.0229,Y -128.1133,Z 159,A -72.7469,B 23.9219,C -1.0912,E1 24.0002,E2 519.7002} C_DIS
LIN {X 49.5491,Y -126.7914,Z 159,A -71.0107,B 23.9215,C -1.1014,E1 24.0048,E2 517.9428} C_DIS
LIN {X 53.0414,Y -125.3719,Z 159,A -69.3665,B 23.9213,C -1.1068,E1 24.0091,E2 516.2893} C_DIS
LIN {X 56.7429,Y -123.7397,Z 159,A -67.1604,B 23.9199,C -1.1366,E1 24.0148,E2 514.0158} C_DIS
LIN {X 61.1145,Y -121.6414,Z 159,A -65.224,B 23.92,C -1.1343,E1 24.0196,E2 512.0905} C_DIS
LIN {X 64.9137,Y -119.6576,Z 159,A -63.8202,B 23.9209,C -1.1158,E1 24.023,E2 510.7363} C_DIS
LIN {X 69.0656,Y -117.3098,Z 159,A -61.6887,B 23.9204,C -1.1262,E1 24.0282,E2 508.5861} C_DIS
LIN {X 73.5252,Y -114.5674,Z 159,A -59.6432,B 23.9206,C -1.1219,E1 24.033,E2 506.558} C_DIS
LIN {X 77.3959,Y -111.9891,Z 159,A -57.3925,B 23.9197,C -1.1418,E1 24.0383,E2 504.2664} C_DIS
LIN {X 80.3905,Y -109.8592,Z 159,A -56.1246,B 23.9202,C -1.1299,E1 24.041,E2 503.0325} C_DIS
LIN {X 83.9771,Y -107.1424,Z 159,A -54.2663,B 23.9202,C -1.1321,E1 24.0451,E2 501.1758} C_DIS
LIN {X 87.0919,Y -104.6266,Z 159,A -51.9522,B 23.9184,C -1.1703,E1 24.0503,E2 498.7772} C_DIS
LIN {X 91.2456,Y -101.0245,Z 159,A -50.4037,B 23.9201,C -1.1339,E1 24.0533,E2 497.3248} C_DIS
LIN {X 93.9913,Y -98.4746,Z 159,A -48.7035,B 23.9196,C -1.1444,E1 24.0568,E2 495.6061} C_DIS
LIN {X 96.747,Y -95.769,Z 159,A -46.9114,B 23.919,C -1.1575,E1 24.0604,E2 493.7897} C_DIS
LIN {X 100.8359,Y -91.4535,Z 159,A -44.7438,B 23.9195,C -1.1456,E1 24.0645,E2 491.6613} C_DIS
LIN {X 103.3612,Y -88.59,Z 159,A -42.9663,B 23.9189,C -1.1591,E1 24.0678,E2 489.8591} C_DIS
LIN {X 105.7624,Y -85.709,Z 159,A -41.2226,B 23.9183,C -1.1724,E1 24.0709,E2 488.0912} C_DIS
LIN {X 107.7905,Y -83.144,Z 159,A -40.0332,B 23.9186,C -1.1659,E1 24.0729,E2 486.9237} C_DIS
LIN {X 110.4674,Y -79.5534,Z 159,A -38.1832,B 23.9185,C -1.1692,E1 24.0759,E2 485.0749} C_DIS
LIN {X 112.8244,Y -76.1728,Z 159,A -36.473,B 23.9183,C -1.1728,E1 24.0786,E2 483.3647} C_DIS
LIN {X 114.9287,Y -72.9599,Z 159,A -34.264,B 23.9165,C -1.2102,E1 24.0821,E2 481.0756} C_DIS
LIN {X 117.7031,Y -68.3934,Z 159,A -32.5943,B 23.9177,C -1.1848,E1 24.0843,E2 479.4775} C_DIS
LIN {X 119.8677,Y -64.5243,Z 159,A -30.616,B 23.9172,C -1.1965,E1 24.087,E2 477.4812} C_DIS
LIN {X 122.0197,Y -60.3513,Z 159,A -28.8883,B 23.9176,C -1.1888,E1 24.0891,E2 475.7819} C_DIS
LIN {X 123.4684,Y -57.3296,Z 159,A -27.5055,B 23.9174,C -1.1916,E1 24.0908,E2 474.4002} C_DIS
LIN {X 124.8752,Y -54.197,Z 159,A -25.5192,B 23.9158,C -1.226,E1 24.0931,E2 472.3409} C_DIS
LIN {X 126.6569,Y -49.8951,Z 159,A -23.7152,B 23.9159,C -1.2235,E1 24.0949,E2 470.5536} C_DIS
LIN {X 127.9748,Y -46.4073,Z 159,A -22.5379,B 23.9167,C -1.2068,E1 24.096,E2 469.4242} C_DIS
LIN {X 130.0075,Y -40.3668,Z 159,A -19.8057,B 23.9162,C -1.218,E1 24.0984,E2 466.6805} C_DIS
LIN {X 131.0755,Y -36.7472,Z 159,A -18.3287,B 23.9162,C -1.217,E1 24.0995,E2 465.2149} C_DIS
LIN {X 131.9383,Y -33.5177,Z 159,A -16.9526,B 23.9161,C -1.2199,E1 24.1005,E2 463.8402} C_DIS
LIN {X 132.7066,Y -30.3332,Z 159,A -15.5295,B 23.9158,C -1.2268,E1 24.1014,E2 462.4088} C_DIS
LIN {X 133.4138,Y -27.0544,Z 159,A -14.1632,B 23.9156,C -1.2289,E1 24.1022,E2 461.0457} C_DIS
LIN {X 134.0291,Y -23.8202,Z 159,A -12.8136,B 23.9156,C -1.2314,E1 24.1028,E2 459.6982} C_DIS
LIN {X 134.5436,Y -20.7177,Z 159,A -11.5807,B 23.9156,C -1.2308,E1 24.1034,E2 458.4745} C_DIS
LIN {X 134.9942,Y -17.5434,Z 159,A -9.9846,B 23.9147,C -1.2488,E1 24.104,E2 456.844} C_DIS
LIN {X 135.4772,Y -13.3127,Z 159,A -8.2867,B 23.9147,C -1.2495,E1 24.1045,E2 455.1551} C_DIS
LIN {X 135.7902,Y -9.6095,Z 159,A -6.6916,B 23.9143,C -1.2563,E1 24.1048,E2 453.5531} C_DIS
LIN {X 136.0539,Y -4.5877,Z 159,A -3.8751,B 23.912,C -1.3021,E1 24.1051,E2 450.6419} C_DIS
LIN {X 136.1238,Y 1.4277,Z 159,A -2.0557,B 23.9136,C -1.2708,E1 24.1051,E2 448.9105} C_DIS
LIN {X 136.0302,Y 5.1989,Z 159,A -0.2114,B 23.9126,C -1.2903,E1 24.1049,E2 447.0302} C_DIS
LIN {X 135.8331,Y 9.0001,Z 159,A 1.0952,B 23.9132,C -1.2791,E1 24.1047,E2 445.759} C_DIS
LIN {X 135.5233,Y 12.8324,Z 159,A 2.6301,B 23.9132,C -1.2798,E1 24.1043,E2 444.2319} C_DIS
LIN {X 135.1509,Y 16.2928,Z 159,A 4.0673,B 23.913,C -1.283,E1 24.1039,E2 442.7958} C_DIS
LIN {X 134.6574,Y 19.9776,Z 159,A 5.7271,B 23.9125,C -1.2933,E1 24.1032,E2 441.1211} C_DIS
LIN {X 134.0256,Y 23.8398,Z 159,A 7.2493,B 23.9125,C -1.2917,E1 24.1025,E2 439.6122} C_DIS
LIN {X 133.3683,Y 27.278,Z 159,A 8.7264,B 23.9123,C -1.2966,E1 24.1017,E2 438.132} C_DIS
LIN {X 132.509,Y 31.1935,Z 159,A 10.5235,B 23.9117,C -1.3079,E1 24.1006,E2 436.3181} C_DIS
LIN {X 131.5809,Y 34.8947,Z 159,A 12.0189,B 23.9117,C -1.3069,E1 24.0995,E2 434.8342} C_DIS
LIN {X 130.7111,Y 38.0237,Z 159,A 13.5613,B 23.911,C -1.3208,E1 24.0983,E2 433.2672} C_DIS
LIN {X 129.3559,Y 42.4094,Z 159,A 15.675,B 23.9102,C -1.3367,E1 24.0965,E2 431.127} C_DIS
LIN {X 128.1239,Y 45.9937,Z 159,A 16.9208,B 23.911,C -1.3223,E1 24.0954,E2 429.9238} C_DIS
LIN {X 126.8884,Y 49.2996,Z 159,A 18.434,B 23.9106,C -1.3283,E1 24.0938,E2 428.4048} C_DIS
LIN {X 125.0775,Y 53.7291,Z 159,A 20.2695,B 23.9108,C -1.3245,E1 24.0919,E2 426.5892} C_DIS
LIN {X 123.6758,Y 56.8812,Z 159,A 21.6349,B 23.9108,C -1.324,E1 24.0903,E2 425.2328} C_DIS
LIN {X 121.2426,Y 61.8979,Z 159,A 24.1298,B 23.9101,C -1.3387,E1 24.0872,E2 422.7158} C_DIS
LIN {X 119.5612,Y 65.0904,Z 159,A 25.6861,B 23.9098,C -1.345,E1 24.0852,E2 421.1527} C_DIS
LIN {X 117.4248,Y 68.8698,Z 159,A 27.4888,B 23.9096,C -1.3487,E1 24.0827,E2 419.3508} C_DIS
LIN {X 115.377,Y 72.2489,Z 159,A 29.1732,B 23.9093,C -1.3543,E1 24.0802,E2 417.6615} C_DIS
LIN {X 113.8659,Y 74.6075,Z 159,A 31.693,B 23.9051,C -1.4309,E1 24.0761,E2 414.9667} C_DIS
LIN {X 108.4181,Y 82.3244,Z 159,A 34.512,B 23.908,C -1.3773,E1 24.0716,E2 412.2935} C_DIS
LIN {X 106.409,Y 84.9045,Z 159,A 35.6604,B 23.9085,C -1.3684,E1 24.0696,E2 411.1727} C_DIS
LIN {X 103.4953,Y 88.4334,Z 159,A 37.5486,B 23.9084,C -1.3709,E1 24.0662,E2 409.2874} C_DIS
LIN {X 100.0034,Y 92.3636,Z 159,A 39.7704,B 23.9081,C -1.3765,E1 24.062,E2 407.0622} C_DIS
LIN {X 97.007,Y 95.5056,Z 159,A 41.6185,B 23.9078,C -1.3817,E1 24.0584,E2 405.2098} C_DIS
LIN {X 93.3203,Y 99.1108,Z 159,A 43.7012,B 23.9078,C -1.3817,E1 24.0543,E2 403.1363} C_DIS
LIN {X 90.4077,Y 101.7751,Z 159,A 45.428,B 23.9074,C -1.3885,E1 24.0507,E2 401.3998} C_DIS
LIN {X 82.0399,Y 108.6327,Z 159,A 49.7181,B 23.9077,C -1.383,E1 24.0415,E2 397.1402} C_DIS
LIN {X 78.5863,Y 111.1568,Z 159,A 51.7175,B 23.907,C -1.3968,E1 24.0368,E2 395.1145} C_DIS
LIN {X 75.1522,Y 113.5073,Z 159,A 53.4985,B 23.9067,C -1.4012,E1 24.0327,E2 393.3287} C_DIS
LIN {X 71.5608,Y 115.8053,Z 159,A 55.3203,B 23.9065,C -1.4055,E1 24.0284,E2 391.5025} C_DIS
LIN {X 67.1226,Y 118.4328,Z 159,A 57.4758,B 23.9064,C -1.4079,E1 24.0232,E2 389.3479} C_DIS
LIN {X 63.5347,Y 120.3931,Z 159,A 58.9803,B 23.9069,C -1.399,E1 24.0195,E2 387.87} C_DIS
LIN {X 60.8658,Y 121.7659,Z 159,A 60.4472,B 23.9062,C -1.4113,E1 24.0158,E2 386.3769} C_DIS
LIN {X 57.4673,Y 123.4048,Z 159,A 61.9185,B 23.9064,C -1.4071,E1 24.0121,E2 384.9199} C_DIS
LIN {X 54.2116,Y 124.8689,Z 159,A 64.15,B 23.9041,C -1.4473,E1 24.0062,E2 382.5952} C_DIS
LIN {X 48.9811,Y 127.0122,Z 159,A 65.8973,B 23.9059,C -1.4164,E1 24.0019,E2 380.928} C_DIS
LIN {X 45.2227,Y 128.3997,Z 159,A 67.5628,B 23.9059,C -1.4169,E1 23.9975,E2 379.2649} C_DIS
LIN {X 41.5629,Y 129.629,Z 159,A 69.0375,B 23.9062,C -1.4105,E1 23.9936,E2 377.8089} C_DIS
LIN {X 38.1938,Y 130.6613,Z 159,A 70.579,B 23.906,C -1.4146,E1 23.9895,E2 376.26} C_DIS
LIN {X 35.1378,Y 131.5161,Z 159,A 71.9325,B 23.9059,C -1.4165,E1 23.9858,E2 374.9043} C_DIS
LIN {X 31.1523,Y 132.519,Z 159,A 73.7641,B 23.9055,C -1.4227,E1 23.9808,E2 373.06} C_DIS
LIN {X 27.3139,Y 133.361,Z 159,A 75.3357,B 23.9057,C -1.4193,E1 23.9765,E2 371.499} C_DIS
LIN {X 23.3587,Y 134.1117,Z 159,A 77.1034,B 23.9055,C -1.4237,E1 23.9717,E2 369.7224} C_DIS
LIN {X 19.6806,Y 134.6998,Z 159,A 78.6014,B 23.9056,C -1.4207,E1 23.9676,E2 368.2335} C_DIS
LIN {X 16.1131,Y 135.1724,Z 159,A 80.079,B 23.9057,C -1.4191,E1 23.9635,E2 366.761} C_DIS
LIN {X 11.8677,Y 135.6117,Z 159,A 82.209,B 23.9048,C -1.4364,E1 23.9574,E2 364.5896} C_DIS
LIN {X 8.3528,Y 135.8729,Z 159,A 83.4517,B 23.9055,C -1.4241,E1 23.9541,E2 363.3778} C_DIS
LIN {X 4.0253,Y 136.0702,Z 159,A 85.1946,B 23.9057,C -1.4199,E1 23.9492,E2 361.6457} C_DIS
LIN {X 0.7228,Y 136.1276,Z 159,A 86.8752,B 23.9049,C -1.4345,E1 23.9444,E2 359.9293} C_DIS
LIN {X -2.7422,Y 136.1027,Z 159,A 88.0603,B 23.9057,C -1.4202,E1 23.9412,E2 358.7794} C_DIS
LIN {X -6.6748,Y 135.9658,Z 159,A 89.6514,B 23.9059,C -1.4164,E1 23.9368,E2 357.1974} C_DIS
LIN {X -10.0013,Y 135.7616,Z 159,A 91.1105,B 23.9058,C -1.4187,E1 23.9327,E2 355.7321} C_DIS
LIN {X -14.132,Y 135.3945,Z 159,A 92.9139,B 23.9056,C -1.4207,E1 23.9277,E2 353.9227} C_DIS
LIN {X -17.8796,Y 134.9502,Z 159,A 94.4454,B 23.9059,C -1.4169,E1 23.9235,E2 352.3994} C_DIS
LIN {X -21.9357,Y 134.3511,Z 159,A 96.1608,B 23.9059,C -1.4152,E1 23.9188,E2 350.6867} C_DIS
LIN {X -25.5575,Y 133.7086,Z 159,A 97.715,B 23.906,C -1.4143,E1 23.9145,E2 349.1329} C_DIS
LIN {X -29.2769,Y 132.9449,Z 159,A 99.4162,B 23.9058,C -1.4181,E1 23.9098,E2 347.4203} C_DIS
LIN {X -33.2844,Y 131.9975,Z 159,A 101.0459,B 23.9062,C -1.4112,E1 23.9054,E2 345.8051} C_DIS
LIN {X -36.2482,Y 131.2151,Z 159,A 102.3062,B 23.9063,C -1.4084,E1 23.902,E2 344.5498} C_DIS
LIN {X -41.4313,Y 129.671,Z 159,A 104.8586,B 23.9057,C -1.4196,E1 23.8951,E2 341.9651} C_DIS
LIN {X -45.9829,Y 128.1278,Z 159,A 106.6337,B 23.9065,C -1.4047,E1 23.8906,E2 340.2231} C_DIS
LIN {X -48.6819,Y 127.1285,Z 159,A 108.0264,B 23.9061,C -1.412,E1 23.8869,E2 338.8092} C_DIS
LIN {X -52.6803,Y 125.5227,Z 159,A 109.6966,B 23.9067,C -1.4024,E1 23.8826,E2 337.1589} C_DIS
LIN {X -56.6223,Y 123.7955,Z 159,A 111.5437,B 23.9067,C -1.4014,E1 23.8779,E2 335.3096} C_DIS
LIN {X -59.9943,Y 122.1959,Z 159,A 113.1045,B 23.9069,C -1.3984,E1 23.874,E2 333.752} C_DIS
LIN {X -63.0655,Y 120.6395,Z 159,A 114.5249,B 23.9071,C -1.3946,E1 23.8705,E2 332.3369} C_DIS
LIN {X -66.7655,Y 118.6339,Z 159,A 116.4017,B 23.907,C -1.3967,E1 23.8658,E2 330.4494} C_DIS
LIN {X -69.8081,Y 116.8695,Z 159,A 118.3228,B 23.9059,C -1.4157,E1 23.8611,E2 328.475} C_DIS
LIN {X -73.7166,Y 114.4449,Z 159,A 120.327,B 23.9059,C -1.4153,E1 23.8564,E2 326.465} C_DIS
LIN {X -77.7553,Y 111.7396,Z 159,A 121.5025,B 23.9085,C -1.3685,E1 23.854,E2 325.4012} C_DIS
LIN {X -82.2737,Y 108.4561,Z 159,A 124.3346,B 23.9075,C -1.387,E1 23.8475,E2 322.5129} C_DIS
LIN {X -86.2349,Y 105.3336,Z 159,A 126.3699,B 23.908,C -1.378,E1 23.843,E2 320.4917} C_DIS
LIN {X -89.5636,Y 102.5182,Z 159,A 127.9664,B 23.9088,C -1.3623,E1 23.8397,E2 318.9277} C_DIS
LIN {X -92.0765,Y 100.2674,Z 159,A 129.621,B 23.9084,C -1.3703,E1 23.8362,E2 317.2462} C_DIS
LIN {X -95.0162,Y 97.4871,Z 159,A 131.3964,B 23.9084,C -1.3697,E1 23.8327,E2 315.4645} C_DIS
LIN {X -98.0497,Y 94.4352,Z 159,A 133.1339,B 23.9089,C -1.3617,E1 23.8293,E2 313.7392} C_DIS
LIN {X -103.8055,Y 88.0685,Z 159,A 136.7537,B 23.9094,C -1.3527,E1 23.8226,E2 310.1247} C_DIS
LIN {X -106.3943,Y 84.923,Z 159,A 138.2274,B 23.9102,C -1.3365,E1 23.82,E2 308.6839} C_DIS
LIN {X -109.499,Y 80.8806,Z 159,A 140.6733,B 23.9098,C -1.3451,E1 23.8159,E2 306.2044} C_DIS
LIN {X -112.0238,Y 77.3462,Z 159,A 142.578,B 23.9098,C -1.3437,E1 23.8128,E2 304.2934} C_DIS
LIN {X -113.9303,Y 74.5096,Z 159,A 144.1072,B 23.9098,C -1.3439,E1 23.8104,E2 302.7555} C_DIS
LIN {X -116.5471,Y 70.3449,Z 159,A 146.0658,B 23.9104,C -1.3326,E1 23.8076,E2 300.8146} C_DIS
LIN {X -118.8612,Y 66.361,Z 159,A 147.9981,B 23.9107,C -1.3265,E1 23.8049,E2 298.8867} C_DIS
LIN {X -120.879,Y 62.6094,Z 159,A 149.8716,B 23.9108,C -1.3251,E1 23.8025,E2 297.0064} C_DIS
LIN {X -122.6668,Y 59.0262,Z 159,A 151.4938,B 23.9112,C -1.317,E1 23.8005,E2 295.395} C_DIS
LIN {X -124.1779,Y 55.7761,Z 159,A 152.9109,B 23.9117,C -1.308,E1 23.7989,E2 293.9921} C_DIS
LIN {X -125.4769,Y 52.7899,Z 159,A 154.3057,B 23.9119,C -1.3049,E1 23.7973,E2 292.5969} C_DIS
LIN {X -126.7361,Y 49.6912,Z 159,A 155.6869,B 23.9121,C -1.2992,E1 23.7959,E2 291.2216} C_DIS
LIN {X -127.94,Y 46.5038,Z 159,A 157.2256,B 23.9121,C -1.2997,E1 23.7944,E2 289.6725} C_DIS
LIN {X -130.1779,Y 39.8103,Z 159,A 160.1592,B 23.9127,C -1.2885,E1 23.7919,E2 286.7491} C_DIS
LIN {X -131.1305,Y 36.5506,Z 159,A 161.6117,B 23.9129,C -1.285,E1 23.7908,E2 285.2964} C_DIS
Enddeposition()
END
